	E_CRYO_BIN_CTRL_STATE.ACTIVE_SWITCHING_OFF:
		M_GetStateLabel	:= 'CLOSING...';
	
	E_CRYO_BIN_CTRL_STATE.ERROR:
		M_GetStateLabel	:= 'ERROR';
END_CASE
END_METHOD

METHOD M_SetStatus
VAR_INPUT
	nState:	E_CRYO_BIN_CTRL_STATE;
END_VAR
// Execute the status of the parent FB.
SUPER^.M_SetStatus(nState);


// Handle alarms
M_UpdateAlarms();
END_METHOD

METHOD M_UpdateAlarms
VAR_INPUT
END_VAR
VAR
	stEventEntry : TcEventEntry;
	sText : STRING;
END_VAR
// Array of EventEntry is initialised in the M_Configure method with 
// the alarms defined for the Valve.

fbAlarmHandler(stAlarms := stat.stAlarms);


// Trigger alarms in case of failure.
// The alarms are raised with a rising edge trigger.
// The alarms are cleared with a falling edge trigger.
IF stat.nState = E_CRYO_BIN_CTRL_STATE.ERROR THEN
	IF Actuator.i_nCouplerState <> 8 THEN
		// System not OPERATIONAL or
		// i_nCouplerState not linked to State variable.
		fbAlarmHandler.M_SetAlarm(Tc_Events.CryoValveEventClass.HardwareError);
		stat.sState	:= 'ERROR: System not OPERATIONAL';
	ELSIF Actuator.stat.nLastCommand = E_CRYO_BIN_ACT_CMD.OFF	THEN
		// Valve failed to Close.
		fbAlarmHandler.M_SetAlarm(Tc_Events.CryoValveEventClass.FailureClose);
		stat.sState	:= 'ERROR: Valve failed to CLOSE.';
	ELSIF Actuator.stat.nLastCommand = E_CRYO_BIN_ACT_CMD.ON	THEN
		// Valve failed to Open.
		fbAlarmHandler.M_SetAlarm(Tc_Events.CryoValveEventClass.FailureOpen);
		stat.sState	:= 'ERROR: Valve failed to OPEN.';
	END_IF

END_IF

//
// Clear non-active alarms
// Alarms and their indexes are defined in M_Configure().
// There are three alarms for Valves:
//   0: NOT_OP
//   1: CLOSE failed
//   2: OPEN  failed
//
IF fbAlarmHandler.arrAlarmState[0]  AND  Actuator.i_nCouplerState = 8 THEN
	fbAlarmHandler.M_ClearAlarm(Tc_Events.CryoValveEventClass.HardwareError);
END_IF

IF fbAlarmHandler.arrAlarmState[1]  AND  stat.nState <> E_CRYO_BIN_CTRL_STATE.ERROR THEN
	fbAlarmHandler.M_ClearAlarm(Tc_Events.CryoValveEventClass.FailureClose);
END_IF

IF fbAlarmHandler.arrAlarmState[2] = TRUE  AND  stat.nState <> E_CRYO_BIN_CTRL_STATE.ERROR THEN
	fbAlarmHandler.M_ClearAlarm(Tc_Events.CryoValveEventClass.FailureOpen);
END_IF


fbAlarmHandler.M_ProcessAlarms(
	arrEventEntry := arrEventEntry,
	sEventString := in_sName);
END_METHOD

METHOD M_User_SetAction : INT
VAR_INPUT
END_VAR
// TODO USER
// Set Valve command based on the input parameter in_bEnable.
//
	
IF	stat.nState = E_CRYO_BIN_CTRL_STATE.ACTIVE_OFF  AND in_bEnable THEN
	// Activate the actuator, i.e. open the valve
	M_User_SetAction	:= E_CRYO_BIN_CTRL_ACTION.ON;
ELSIF  stat.nState = E_CRYO_BIN_CTRL_STATE.ACTIVE_ON AND NOT in_bEnable THEN
	// Dectivate the actuator, i.e. close the valve
	M_User_SetAction	:= E_CRYO_BIN_CTRL_ACTION.OFF;
ELSE
	// Don't do anything
	M_User_SetAction	:= E_CRYO_BIN_CTRL_ACTION.NONE;
END_IF
END_METHOD

END_FUNCTION_BLOCK

// ---- POUs/Valve/FB_CRYO_BIN_CTRL.TcPOU
// Binary Controller
FUNCTION_BLOCK FB_CRYO_BIN_CTRL
VAR_INPUT
	in_sName:			STRING := 'Binary Controller';	// Controller name
	in_nFeedback:		E_CRYO_BIN_ACT_FEEDBACK := E_CRYO_BIN_ACT_FEEDBACK.ON_ONLY;	// Feedbacks
	in_nTimeout:		UDINT := 10000;	// Timeout for switching on/off [ms]. Default 10000.
	in_bActiveLowCtrl:	BOOL := FALSE;	// Active Low for Control output
	in_bActiveLowStat:	BOOL := FALSE;	// Active Low for Status signals, i.e. feedback
	in_bEnable:			BOOL := FALSE;	// Controller active while in_bEnable is TRUE
END_VAR
VAR
	
	{attribute 'OPC.UA.DA' := '1'}
	Actuator:	FB_CRYO_BIN_ACT;	// Heater, valve, etc.
	
	{attribute 'OPC.UA.DA' := '1'}
	{attribute 'OPC.UA.DA.Access' := '1'}
	stat:		T_CRYO_BIN_CTRL_STATUS;


	{attribute 'OPC.UA.DA' := '0'}
	bReset:		BOOL := FALSE;		// RESET Command


	{attribute 'OPC.UA.DA' := '0'}
	timer:		TON;		// Timer for commands
	
	// Controller logs
	logs:	FB_CRYO_FUNCTION_LOG;
	
	//
	// Triggers.
	//
	// Capture Enable/Disable.
	trigEnable:		R_TRIG;	// in_bEnable
	trigDisable:	F_TRIG;	// in_bEnable
	// Capture ON/OFF.
	trigON:			R_TRIG;	// i_bIn
	trigOFF:		F_TRIG;	// i_bIn
END_VAR

// Don't do anything until the controller is configured
IF NOT stat.bConfigured THEN
	M_Configure();
	RETURN;
END_IF

// Increment cycle counter
stat.nCycleCounter := stat.nCycleCounter + 1;


// Execute Actuator FB on every cycle
Actuator(
	in_nFeedback		:= in_nFeedback,
	in_nTimeout			:= in_nTimeout,
	in_bActiveLowCtrl	:= in_bActiveLowCtrl,
	in_bActiveLowStat	:= in_bActiveLowStat);


CASE stat.nState OF
	/////////////////////////////////
	E_CRYO_BIN_CTRL_STATE.NONE:
	/////////////////////////////////
	//
	// This is the state on power-up.
	// Determine the initial state based on the command amd actuator state.
	IF Actuator.stat.bError  OR NOT stat.bCtrlOK	THEN
		stat.nState	:= E_CRYO_BIN_CTRL_STATE.ERROR;
	ELSIF in_bEnable  AND  Actuator.stat.bON	THEN
		stat.nState	:= E_CRYO_BIN_CTRL_STATE.ACTIVE_ON;
	ELSIF in_bEnable  AND  Actuator.stat.bOFF	THEN
		stat.nState	:= E_CRYO_BIN_CTRL_STATE.ACTIVE_OFF;
	ELSIF NOT in_bEnable  THEN
		stat.nState	:= E_CRYO_BIN_CTRL_STATE.OFF;
	END_IF
	M_SetStatus(stat.nState);	
	logs.M_LogInfo(M_GetStateLabel(stat.nState));
	RETURN;
	

	/////////////////////////////////
	E_CRYO_BIN_CTRL_STATE.OFF:
	/////////////////////////////////
	//
	IF	Actuator.stat.bError	OR NOT stat.bCtrlOK	THEN
		stat.nState	:= E_CRYO_BIN_CTRL_STATE.ERROR;
	ELSIF in_bEnable  THEN
		// Activate the control loop.
		// Goto Active_Off first.
		//
		// Start the timer
		timer(IN:=FALSE);
		timer(IN:=TRUE, PT:=UDINT_TO_TIME(in_nTimeout));
		// Set next state
		stat.nState	:= E_CRYO_BIN_CTRL_STATE.ACTIVE_OFF;
	END_IF
	M_SetStatus(stat.nState);	
	RETURN;
	
	
	/////////////////////////////////
	E_CRYO_BIN_CTRL_STATE.ACTIVE_OFF:
	/////////////////////////////////
	//
	IF	Actuator.stat.bError	OR NOT stat.bCtrlOK  THEN
		stat.nState	:= E_CRYO_BIN_CTRL_STATE.ERROR;
	ELSIF NOT in_bEnable  THEN
		// Goto Off.
		//
		// Set next state
		stat.nState	:= E_CRYO_BIN_CTRL_STATE.OFF;
	ELSIF M_User_SetAction() = E_CRYO_BIN_CTRL_ACTION.ON THEN
		// Goto Active_Off.
		//
		// Start the timer
		timer(IN:=FALSE);
		timer(IN:=TRUE, PT:=UDINT_TO_TIME(in_nTimeout));
		
		// Trigger action
		Actuator(in_bExecute:=FALSE);
		Actuator(in_bExecute:=TRUE, in_nCommand:=E_CRYO_BIN_ACT_CMD.ON);
		
		// Set next state
		stat.nState	:= E_CRYO_BIN_CTRL_STATE.ACTIVE_SWITCHING_ON;
		logs.M_LogInfo(M_GetStateLabel(stat.nState));
	END_IF
	M_SetStatus(stat.nState);	
	RETURN;
	
	
	//////////////////////////////////////////
	E_CRYO_BIN_CTRL_STATE.ACTIVE_SWITCHING_ON:
	//////////////////////////////////////////
	//
	// Check for timeout
	timer(IN:=TRUE);
	IF timer.Q THEN
		// Stop the timer
		timer(IN:=FALSE);
		// Goto ERROR state
		stat.nState	:= E_CRYO_BIN_CTRL_STATE.ERROR;
	ELSIF	Actuator.stat.bError	THEN
		stat.nState	:= E_CRYO_BIN_CTRL_STATE.ERROR;
	ELSIF Actuator.stat.bON THEN
		// The actuator is ON, transition completed.
		// Goto Active_On.
		stat.nState	:= E_CRYO_BIN_CTRL_STATE.ACTIVE_ON;
		logs.M_LogInfo(M_GetStateLabel(stat.nState));
	END_IF
	M_SetStatus(stat.nState);	
	RETURN;
	

	/////////////////////////////////
	E_CRYO_BIN_CTRL_STATE.ACTIVE_ON:
	/////////////////////////////////
	//
	IF	Actuator.stat.bError	THEN
		stat.nState	:= E_CRYO_BIN_CTRL_STATE.ERROR;
	ELSIF	NOT in_bEnable 		OR  
			NOT stat.bCtrlOK	OR
			M_User_SetAction() = E_CRYO_BIN_CTRL_ACTION.OFF THEN
		// Goto Active_Off.
		// If NOT in_bExecute, the system will continue to complete OFF
		//
		// Start the timer
		timer(IN:=FALSE);
		timer(IN:=TRUE, PT:=UDINT_TO_TIME(in_nTimeout));
		
		// Trigger action
		Actuator(in_bExecute:=FALSE);
		Actuator(in_bExecute:=TRUE, in_nCommand:=E_CRYO_BIN_ACT_CMD.OFF);
		
		// Set next state
		stat.nState	:= E_CRYO_BIN_CTRL_STATE.ACTIVE_SWITCHING_OFF;
		logs.M_LogInfo(M_GetStateLabel(stat.nState));
	END_IF
	M_SetStatus(stat.nState);	
	RETURN;
	
	
	///////////////////////////////////////////
	E_CRYO_BIN_CTRL_STATE.ACTIVE_SWITCHING_OFF:
	///////////////////////////////////////////
	//
	// Check for timeout
	timer(IN:=TRUE);
	IF timer.Q THEN
		// Stop the timer
		timer(IN:=FALSE);
		// Goto ERROR state
		stat.nState	:= E_CRYO_BIN_CTRL_STATE.ERROR;
	ELSIF	Actuator.stat.bError	THEN
		stat.nState	:= E_CRYO_BIN_CTRL_STATE.ERROR;
	ELSIF Actuator.stat.bOFF THEN
		// The actuator is OFF, transition completed.
		// Goto Active_Off.
		stat.nState	:= E_CRYO_BIN_CTRL_STATE.ACTIVE_OFF;
		logs.M_LogInfo(M_GetStateLabel(stat.nState));
	END_IF
	M_SetStatus(stat.nState);	
	RETURN;
	
	/////////////////////////////////
	E_CRYO_BIN_CTRL_STATE.ERROR:
	/////////////////////////////////
	//
	M_User_TryRecovery();

END_CASE

METHOD M_Configure
VAR_INPUT
END_VAR
// Overwrite this method for specific implementation.
// Here we have just a dummy implementation to set
// stat.bConfigured	:= TRUE;


// Device specific implementation
// TODO


// A MUST !!!

// This call just configures logs at the very start.
// Logging is done by explicit calls to M_LogInfo().
logs(in_sName := in_sName);

stat.bConfigured	:= TRUE;
END_METHOD

// Set labels for logging.
// Examples:
//	ON, OFF (for heaters)
//	OPEN, CLOSE (for valves)
METHOD M_GetStateLabel : STRING
VAR_INPUT
	state:	E_CRYO_BIN_CTRL_STATE;
END_VAR
CASE state OF
	E_CRYO_BIN_CTRL_STATE.OFF:
		M_GetStateLabel	:= 'OFF';
	
	E_CRYO_BIN_CTRL_STATE.ACTIVE_SWITCHING_ON:
		M_GetStateLabel	:= 'SWITCHING_ON';
	
	E_CRYO_BIN_CTRL_STATE.ACTIVE_OFF:
		M_GetStateLabel	:= 'OFF';
	
	E_CRYO_BIN_CTRL_STATE.ACTIVE_ON:
		M_GetStateLabel	:= 'ON';
	
	E_CRYO_BIN_CTRL_STATE.ACTIVE_SWITCHING_OFF:
		M_GetStateLabel	:= 'SWITCHING_OFF';
	
	E_CRYO_BIN_CTRL_STATE.ERROR:
		M_GetStateLabel	:= 'ERROR';
END_CASE
END_METHOD

METHOD M_Reset
VAR_INPUT
END_VAR
// By setting the bReset flag,
// The actuator will try to exit error state.
// In ERROR state, method M_User_TryRecovery() is executed.
bReset	:= TRUE;
END_METHOD

METHOD M_SetStatus
VAR_INPUT
	nState:	E_CRYO_BIN_CTRL_STATE;
END_VAR
stat.bActON		:= Actuator.stat.bON;
stat.bActOFF	:= Actuator.stat.bOFF;


CASE nState OF
	
	E_CRYO_BIN_CTRL_STATE.OFF:
	stat.bDone	:= TRUE;
	stat.bBusy	:= FALSE;
	stat.bError	:= FALSE;
	stat.bActive:= FALSE;
	stat.sState	:= 'OFF';
	
	E_CRYO_BIN_CTRL_STATE.ACTIVE_OFF:
	stat.bDone	:= TRUE;
	stat.bBusy	:= FALSE;
	stat.bError	:= FALSE;
	stat.bActive:= TRUE;
	stat.sState	:= 'ACTIVE_OFF';
	
	E_CRYO_BIN_CTRL_STATE.ACTIVE_ON:
	stat.bDone	:= TRUE;
	stat.bBusy	:= FALSE;
	stat.bError	:= FALSE;
	stat.bActive:= TRUE;
	stat.sState	:= 'ACTIVE_ON';
	
	E_CRYO_BIN_CTRL_STATE.ACTIVE_SWITCHING_ON:
	stat.bDone	:= FALSE;
	stat.bBusy	:= TRUE;
	stat.bError	:= FALSE;
	stat.bActive:= TRUE;
	stat.sState	:= 'ACTIVE_SWITCHING_ON...';
	
	E_CRYO_BIN_CTRL_STATE.ACTIVE_SWITCHING_OFF:
	stat.bDone	:= FALSE;
	stat.bBusy	:= TRUE;
	stat.bError	:= FALSE;
	stat.bActive:= TRUE;
	stat.sState	:= 'ACTIVE_SWITCHING_OFF...';
	
	E_CRYO_BIN_CTRL_STATE.ERROR:
	stat.bDone	:= TRUE;
	stat.bBusy	:= FALSE;
	stat.bError	:= TRUE;
	stat.bActive:= FALSE;
	stat.sState	:= 'ERROR';

END_CASE
END_METHOD

METHOD M_User_SetAction : INT
VAR_INPUT
END_VAR
// TODO USER
//
// This method implements the logic for controlling the actuator.
// The actuator can be a heater, valve, etc.
//
// This example implements the heater control with the following assumptions:
// There are two input values from sensors and two deltas for comparison.
//
// in_lrInput1 - Temperature of the Cryo Bench (B)
// in_lrInput2 - Temperature of the Detector (D). Coming from Lakeshore.
// in_lrPar1 - Delta [K] to turn the heater ON:  IF B < D - in_lrPar1
// in_lrPar2 - Delta [K] to turn the heater OFF: IF B > D - in_lrPar2
//
// in_lrDelta1 > in_lrDelta2, e.g. 10K > 4K.
//
IF	stat.nState = E_CRYO_BIN_CTRL_STATE.ACTIVE_OFF  OR  
	stat.nState = E_CRYO_BIN_CTRL_STATE.ACTIVE_ON THEN
(*	
	IF in_lrInput1 < in_lrInput2 - in_lrPar1 THEN
		// Activate the actuator
		M_User_SetOutput	:= E_CRYO_BIN_CTRL_ACTION.ON;
	ELSIF in_lrInput1 > in_lrInput2 - in_lrPar2 THEN
		// Dectivate the actuator
		M_User_SetOutput	:= E_CRYO_BIN_CTRL_ACTION.OFF;
	END_IF
*)
ELSE
	// Don't do anything
	M_User_SetAction	:= E_CRYO_BIN_CTRL_ACTION.NONE;
END_IF
END_METHOD

METHOD M_User_TryRecovery
VAR_INPUT
END_VAR
// TODO USER
// This is the default recovery routine.
// To be customided by the user, if needed.
//
IF bReset THEN
	// RESET the controller in order to try to clear error
	bReset	:= FALSE;	// Clear RESET flag
	
	// Start the timer
	timer(IN:=FALSE);
	timer(IN:=TRUE, PT:=T#5S);
	
	// Trigger action
	Actuator(in_bExecute:=FALSE);
	Actuator(in_bExecute:=TRUE, in_nCommand:=E_CRYO_BIN_ACT_CMD.OFF);
	
	// Goto SWITCHING_OFF state
	stat.nState	:= E_CRYO_BIN_CTRL_STATE.ACTIVE_SWITCHING_OFF;
	M_SetStatus(stat.nState);	
ELSIF NOT Actuator.stat.bError AND stat.bCtrlOK  THEN
	// Self recovery since everything seems to be OK now.
	// Goto NONE state.
	// From there proper state will be found and set.
	stat.nState	:= E_CRYO_BIN_CTRL_STATE.NONE;
	M_SetStatus(stat.nState);	
END_IF
END_METHOD

END_FUNCTION_BLOCK

// ---- POUs/Services/FB_SERVICES.TcPOU
FUNCTION_BLOCK FB_SERVICES
VAR_INPUT
END_VAR
VAR_OUTPUT
END_VAR
VAR    
    // Let's always link the EtherCAT DevState, so that 
    // we always have one sync variable (even if all subsystems are disabled)
    {attribute 'TcLinkTo' := 'TIID^Device 1 (EtherCAT)^Inputs^DevState'}
	i_nDevState AT %I* : UINT;
    
    {attribute 'TcLinkTo' := '.i_inTime             := TIID^Device 1 (EtherCAT)^PLC (EK1200)^PTP (EL6688)^  External Sync^Internal time stamp;
                              .i_exTime             := TIID^Device 1 (EtherCAT)^PLC (EK1200)^PTP (EL6688)^  External Sync^External time stamp;
                              .i_dc2TcOffset        := TIID^Device 1 (EtherCAT)^InfoData^DcToTcTimeOffset;
                              .i_dc2ExtOffset       := TIID^Device 1 (EtherCAT)^InfoData^DcToExtTimeOffset;
                              .i_extDevNotConnected := TIID^Device 1 (EtherCAT)^PLC (EK1200)^PTP (EL6688)^  External Sync^External device not connected;
                              .i_AdsAddr            := TIID^Device 1 (EtherCAT)^PLC (EK1200)^PTP (EL6688)^InfoData^AdsAddr;
                              .i_exNtpExtTime       := TIRC^TcCOM Objects^NtpProvider^Outputs^nExtTime;
                              .i_exNtpSysTime       := TIRC^TcCOM Objects^NtpProvider^Outputs^nSysTime;
                              .i_exNtpExtOffset     := TIRC^TcCOM Objects^NtpProvider^Outputs^nSysToExtTimeOffset;
                              .i_NtpConnected       := TIRC^TcCOM Objects^NtpProvider^Diagnostic^bIsConnected;
                              .i_exNtpSynchronized  := TIRC^TcCOM Objects^NtpProvider^Diagnostic^bIsSynchronized'}
    fbTime : FB_TIME;

END_VAR

fbTime();

END_FUNCTION_BLOCK

// ---- HMI/PRG_HMI.TcPOU
{attribute 'OPC.UA.DA' := '0'}
PROGRAM PRG_HMI
VAR
    // System health & busy status
    fbHealthStatus: 		FB_HMI_HEALTH_STATUS;
    fbBusyStatus: 			FB_HMI_BUSY_STATUS;
    fbStatusColor: 			T_HMI_COLORS;
    
    // BUTTONS
    // ===============================================================================================
    
    // buttons at the main screen
    fbHomeButton: 			FB_HMI_BUTTON('Home'     , 		'Start'      , 	E_HMI_TABS.HOME);
    fbServicesButton : 		FB_HMI_BUTTON('Services' , 		'Services'   , 	E_HMI_TABS.SERVICES);	
	fbEventsButton: 		FB_HMI_BUTTON('Events' , 		'Events', 		E_HMI_TABS.EVENTS);
	fbCryoInterlocksButton: FB_HMI_BUTTON('Cryo Interlocks' ,'Interlock', 	E_HMI_TABS.CRYO_INTERLOCKS);
	
	// ICS Subsystem buttons
	fbShuttersButton: 		FB_HMI_BUTTON('Shutters' , 		'', 			E_HMI_TABS.SHUTTERS);
	fbTipTiltButton: 		FB_HMI_BUTTON('Tip Tilt' , 		'', 			E_HMI_TABS.TIP_TILT);
	fbDelayLinesButton: 	FB_HMI_BUTTON('Delay Lines' , 	'', 			E_HMI_TABS.DELAY_LINES);
	fbCO2TransStagesButton: FB_HMI_BUTTON('CO2 Translation','', 			E_HMI_TABS.CO2_TRANSLATION_STAGES);
	fbZnSeActuatorsButton: 	FB_HMI_BUTTON('ZnSe Actuators' ,'', 			E_HMI_TABS.ZNSE_ACTUATORS);
	fbBirefringenceButton: 	FB_HMI_BUTTON('Birefringence' , '', 			E_HMI_TABS.BIREFRINGENCE_ACTUATORS);
	fbBeamSplitterButton: 	FB_HMI_BUTTON('Beam Splitter' , '', 			E_HMI_TABS.CALIBRATION_UNIT_BEAM_SPLITER);
	fbCO2PressureButton: 	FB_HMI_BUTTON('CO2 Pressure' , 	'', 			E_HMI_TABS.CO2_PRESSURE_CONTROL);
	
    // COMPONENTS
    // ===============================================================================================

    {attribute 'OPC.UA.DA' := '0'}
    fbServices: 			FB_HMI_SERVICES;
	{attribute 'OPC.UA.DA' := '0'}
	fbEvents: 				FB_HMI_EVENTS;
	{attribute 'OPC.UA.DA' := '0'}
	fbCryoInterlocks: 		FB_HMI_CRYO_INTERLOCKS;
	
	{attribute 'OPC.UA.DA' := '0'}
	fbShutters:				FB_HMI_SHUTTERS;
	{attribute 'OPC.UA.DA' := '0'}	
	fbTipTilt:				FB_HMI_TIP_TILT;
	{attribute 'OPC.UA.DA' := '0'}
	fbDelayLines:	        FB_HMI_DELAY_LINES;
	{attribute 'OPC.UA.DA' := '0'}
	fbCO2TransStages:       FB_HMI_CO2_TRANS_STAGES;
	{attribute 'OPC.UA.DA' := '0'}
	fbZnSeActuators:        FB_HMI_ZNSE_ACTUATORS;
	{attribute 'OPC.UA.DA' := '0'}
	fbBirefringence:	    FB_HMI_BIREFRINGENCE;
	{attribute 'OPC.UA.DA' := '0'}
	fbBeamSplitter:         FB_HMI_CALIBRATION_BEAM_SPLITTER;
	{attribute 'OPC.UA.DA' := '0'}
	fbCO2Pressure:          FB_HMI_CO2_PRESSURE_CONTROL;

    
    // active tab of the main frame
    eActiveTab : E_HMI_TABS := E_HMI_TABS.HOME;
    sActiveName : STRING;
END_VAR

//// update the components
fbServices(fbInstance := MAIN.fbServices);
fbEvents(); 				
fbCryoInterlocks(fbInstance := MAIN.nott_ics.Cryo_Interlocks); 		

// SubSystems
fbShutters(fbInstance := MAIN.nott_ics.Shutters);			
fbTipTilt(fbInstance := MAIN.nott_ics.TipTilt);		
fbDelayLines(fbInstance := MAIN.nott_ics.Delay_Lines);			
fbCO2TransStages(fbInstance := MAIN.nott_ics.CO2TransStages);					
fbZnSeActuators(fbInstance := MAIN.nott_ics.ZnSeActuators);	 		
fbBirefringence(fbInstance := MAIN.nott_ics.Birefringence);		
fbBeamSplitter(fbInstance := MAIN.nott_ics.Calibration_Unit_Beam_Splitter);				
fbCO2Pressure(fbInstance := MAIN.nott_ics.CO2_Pressure_Control);

// update the status
M_UpdateStatus();

// update the system-level buttons
fbHomeButton(stColor := fbStatusColor, nActiveTab := eActiveTab, sActiveName := sActiveName);
// buttons at the main screen 
fbServicesButton(stColor := fbServices.fbStatusColor, nActiveTab := eActiveTab, sActiveName := sActiveName);	
fbEventsButton(stColor:= fbEvents.fbStatusColor, nActiveTab:= eActiveTab, sActiveName:= sActiveName);		
fbCryoInterlocksButton(stColor:= fbCryoInterlocks.fbStatusColor, nActiveTab:= eActiveTab, sActiveName:= sActiveName); 	

fbShuttersButton(stColor:= fbShutters.fbStatusColor, nActiveTab:= eActiveTab, sActiveName:= sActiveName); 			
fbTipTiltButton(stColor:= fbTipTilt.fbStatusColor, nActiveTab:= eActiveTab, sActiveName:= sActiveName); 		
fbDelayLinesButton(stColor:= fbDelayLines.fbStatusColor, nActiveTab:= eActiveTab, sActiveName:= sActiveName); 	
fbCO2TransStagesButton(stColor:= fbCO2TransStages.fbStatusColor, nActiveTab:= eActiveTab, sActiveName:= sActiveName); 				
fbZnSeActuatorsButton(stColor:= fbZnSeActuators.fbStatusColor, nActiveTab:= eActiveTab, sActiveName:= sActiveName); 		
fbBirefringenceButton(stColor:= fbBirefringence.fbStatusColor, nActiveTab:= eActiveTab, sActiveName:= sActiveName); 		
fbBeamSplitterButton(stColor:= fbBeamSplitter.fbStatusColor, nActiveTab:= eActiveTab, sActiveName:= sActiveName); 			
fbCO2PressureButton(stColor:= fbCO2Pressure.fbStatusColor, nActiveTab:= eActiveTab, sActiveName:= sActiveName);

METHOD M_UpdateStatus
VAR_INPUT
END_VAR
// update the health & busy statuses
//fbHealthStatus(
//    bIsEnabled :=   fbImg.fbHealthStatus.bEnabled
//                AND fbSca.fbHealthStatus.bEnabled,
//    bIsGood :=      fbImg.fbHealthStatus.bGood
//                AND fbSca.fbHealthStatus.bGood);
              //AND fbServices.fbHealthStatus.bGood
              //AND fbLms.fbHealthStatus.bGood (* AND ... *));
//fbBusyStatus(
//    bIsEnabled :=   fbImg.fbBusyStatus.bEnabled
//                AND fbSca.fbBusyStatus.bEnabled,
//    bIsBusy := fbServices.fbBusyStatus.bBusy 
//                 OR fbImg.fbBusyStatus.bBusy 
//                 OR fbLms.fbBusyStatus.bBusy 
//                 OR fbSca.fbBusyStatus.bBusy);

fbStatusColor := F_HMI_HEALTH_BUSY_TO_COLOR(fbHealthStatus, fbBusyStatus);
END_METHOD

END_PROGRAM

// ---- HMI/POUs/Services/Status/FB_HMI_HEALTH_STATUS.TcPOU
FUNCTION_BLOCK FB_HMI_HEALTH_STATUS
VAR_INPUT
	// TRUE if the subject is in Good health
	bIsGood: BOOL;
	// TRUE to add a warning to the Good health state
	bHasWarning: BOOL := FALSE;
	// TRUE if the health status is used
	bIsEnabled: BOOL := TRUE;
END_VAR
VAR_OUTPUT
	// TRUE if the subject is enabled
	bEnabled: BOOL;
    // TRUE if the subject is in good health
	bGood: BOOL;
	// TRUE if the subject is in good health, but there are one or more warnings present
	bWarning: BOOL;
	// TRUE if the subject is in bad health
	bBad: BOOL;
END_VAR
VAR_IN_OUT
END_VAR
VAR
END_VAR

bEnabled := bIsEnabled;
bBad := (NOT(bIsGood)) AND bIsEnabled;
bGood := (bIsGood AND (NOT(bHasWarning))) AND bIsEnabled;
bWarning := (bIsGood AND bHasWarning) AND bIsEnabled;

END_FUNCTION_BLOCK

// ---- HMI/POUs/Services/Status/FB_HMI_BUSY_STATUS.TcPOU
FUNCTION_BLOCK FB_HMI_BUSY_STATUS
VAR_INPUT
	// TRUE if busy
	bIsBusy: BOOL;
	// TRUE if the busy status is used
	bIsEnabled: BOOL := TRUE;
END_VAR
VAR_OUTPUT
	// TRUE if the subject is enabled
	bEnabled: BOOL;
	///The subject is idle
	bIdle: BOOL;
	///The subject is busy
	bBusy: BOOL;
END_VAR
VAR_IN_OUT
END_VAR
VAR
END_VAR

bBusy := bIsBusy AND bIsEnabled;
bIdle := (NOT(bIsBusy)) AND bIsEnabled;

END_FUNCTION_BLOCK

// ---- HMI/POUs/Util/Button/FB_HMI_BUTTON.TcPOU
FUNCTION_BLOCK FB_HMI_BUTTON
VAR_INPUT
    stColor : T_HMI_COLORS;
END_VAR
VAR_IN_OUT
    nActiveTab : INT;
    sActiveName : STRING;
END_VAR
VAR_OUTPUT
    sName : STRING;
    sIconName : STRING;
    nThisTab : INT;
    bActivated : BOOL;
    bNotActivated : BOOL;
    
    bIsNotGreen : BOOL;
    bIsNotRed : BOOL;
    bIsNotBlue : BOOL;
    bIsNotOrange : BOOL;
    bIsNotGray : BOOL;
END_VAR
VAR
    bDoActivate : BOOL;
    bPreviouslyActive : BOOL;
END_VAR

IF bDoActivate THEN
    nActiveTab := nThisTab;
    bDoActivate := FALSE;
END_IF

bActivated := nActiveTab = nThisTab;
bNotActivated := NOT bActivated;

IF bActivated AND NOT bPreviouslyActive THEN
    sActiveName := sName;
    bPreviouslyActive := TRUE;
END_IF

IF bNotActivated THEN
    bPreviouslyActive := FALSE;
END_IF

bIsNotRed    := stColor.bg <> E_HMI_Colors.RED;
bIsNotBlue   := stColor.bg <> E_HMI_Colors.BLUE;
bIsNotOrange := stColor.bg <> E_HMI_Colors.ORANGE;
bIsNotGray   := stColor.bg <> E_HMI_Colors.GRAY;
bIsNotGreen  := stColor.bg <> E_HMI_Colors.GREEN;

METHOD FB_init : BOOL
VAR_INPUT
	bInitRetains : BOOL; // if TRUE, the retain variables are initialized (warm start / cold start)
	bInCopyCode : BOOL;  // if TRUE, the instance afterwards gets moved into the copy code (online change)
    sName : STRING;
    sIconName : STRING;
    nThisTab : INT;
END_VAR
THIS^.sName := sName;
THIS^.sIconName := sIconName;
THIS^.nThisTab := nThisTab;
END_METHOD

METHOD M_SetIconName
VAR_INPUT
    sIconName : STRING;
END_VAR
THIS^.sIconName := sIconName;
END_METHOD

END_FUNCTION_BLOCK

// ---- HMI/POUs/Services/FB_HMI_SERVICES.TcPOU
FUNCTION_BLOCK FB_HMI_SERVICES EXTENDS FB_HMI_COMPONENT
VAR_INPUT
END_VAR
VAR_OUTPUT
END_VAR
VAR_IN_OUT
    fbInstance : FB_SERVICES;
END_VAR
VAR
    fbTime : FB_HMI_SERVICES_TIME;
END_VAR

fbTime(fbInstance := fbInstance.fbTime);

fbHealthStatus(
    bIsEnabled  := fbTime.fbHealthStatus.bEnabled,
    bIsGood     := fbTime.fbHealthStatus.bGood);
fbBusyStatus(
    bIsEnabled  := fbTime.fbBusyStatus.bEnabled,
    bIsBusy     := fbTime.fbBusyStatus.bBusy);

M_UpdateStatusColor();

END_FUNCTION_BLOCK

// ---- HMI/POUs/Util/Component/FB_HMI_COMPONENT.TcPOU
FUNCTION_BLOCK FB_HMI_COMPONENT
VAR_INPUT
END_VAR
VAR_OUTPUT
    fbHealthStatus : FB_HMI_HEALTH_STATUS;
    fbBusyStatus : FB_HMI_BUSY_STATUS;
    fbStatusColor : T_HMI_COLORS;
END_VAR
VAR
END_VAR

METHOD PROTECTED M_UpdateStatusColor
VAR_INPUT
END_VAR
// health and busy states must be updated by the subtype before calling this method!
fbStatusColor := F_HMI_HEALTH_BUSY_TO_COLOR(fbHealthStatus, fbBusyStatus);
END_METHOD

END_FUNCTION_BLOCK

// ---- HMI/POUs/Services/Status/F_HMI_HEALTH_BUSY_TO_COLOR.TcPOU
FUNCTION F_HMI_HEALTH_BUSY_TO_COLOR : T_HMI_COLORS
VAR_IN_OUT
    fbHealthStatus : FB_HMI_HEALTH_STATUS;
    fbBusyStatus   : FB_HMI_BUSY_STATUS;
END_VAR
VAR_OUTPUT
END_VAR
VAR
END_VAR

IF fbHealthStatus.bGood THEN
	IF fbBusyStatus.bBusy THEN
		F_HMI_HEALTH_BUSY_TO_COLOR.fg := E_HMI_COLORS.WHITE;
		F_HMI_HEALTH_BUSY_TO_COLOR.bg := E_HMI_COLORS.BLUE;
	ELSE
		F_HMI_HEALTH_BUSY_TO_COLOR.fg := E_HMI_COLORS.BLACK;
		F_HMI_HEALTH_BUSY_TO_COLOR.bg := E_HMI_COLORS.GREEN;
	END_IF
ELSIF fbHealthStatus.bBad THEN
	F_HMI_HEALTH_BUSY_TO_COLOR.fg := E_HMI_COLORS.WHITE;
	F_HMI_HEALTH_BUSY_TO_COLOR.bg := E_HMI_COLORS.RED;
ELSIF fbHealthStatus.bWarning THEN
	F_HMI_HEALTH_BUSY_TO_COLOR.fg := E_HMI_COLORS.WHITE;
	F_HMI_HEALTH_BUSY_TO_COLOR.bg := E_HMI_COLORS.ORANGE;
ELSE
	F_HMI_HEALTH_BUSY_TO_COLOR.fg := E_HMI_COLORS.BLACK;
	F_HMI_HEALTH_BUSY_TO_COLOR.bg := E_HMI_COLORS.GRAY;
END_IF

END_FUNCTION

// ---- HMI/POUs/Services/FB_HMI_SERVICES_TIME.TcPOU
FUNCTION_BLOCK FB_HMI_SERVICES_TIME EXTENDS FB_HMI_COMPONENT
VAR_INPUT
END_VAR
VAR_OUTPUT
END_VAR
VAR_IN_OUT
    fbInstance : FB_TIME;
END_VAR
VAR
    // because GUI_TEMPLATE_TIME is a large height,
    // and because scrolling doesn't seem to work (bug in TC HMI?),
    // we display the GUI_TEMPLATE_TIME twice, with an offset in between 
    nAbsoluteMovementY : INT := -495;
    
    sUtc : STRING;
END_VAR


// update the health & busy states
fbHealthStatus(
    bIsGood     := fbInstance.stat.signal.qos = E_TIME_SIGNAL_QOS.VALID,
    bIsEnabled  := fbInstance.stat.signal.status = E_TIME_SIGNAL_STATUS.CONNECTED);
fbBusyStatus(bIsBusy := FALSE); // never busy

sUtc := LEFT(fbInstance.stat.sUtcTime, 19); 

M_UpdateStatusColor();

END_FUNCTION_BLOCK

// ---- HMI/POUs/Events/FB_HMI_EVENTS.TcPOU
FUNCTION_BLOCK FB_HMI_EVENTS EXTENDS FB_HMI_COMPONENT
VAR_INPUT
END_VAR
VAR_OUTPUT
END_VAR

END_FUNCTION_BLOCK

// ---- HMI/POUs/CRYO_Interlocks/FB_HMI_CRYO_INTERLOCKS.TcPOU
FUNCTION_BLOCK FB_HMI_CRYO_INTERLOCKS EXTENDS FB_HMI_COMPONENT
VAR_INPUT
END_VAR
VAR_OUTPUT
END_VAR
VAR
END_VAR
VAR_IN_OUT
	{attribute 'OPC.UA.DA' := '0'}
	fbInstance		: FB_NOTT_CRYO_INTERLOCKS;


END_VAR

fbHealthStatus( 
				bIsEnabled:= TRUE, 
				bIsGood := NOT fbInstance.stat.bError,
				bHasWarning := fbInstance.stat.bWarning
				);
				
fbBusyStatus(
				bIsBusy := fbInstance.stat.bBusy,
				bIsEnabled := TRUE);				
M_UpdateStatusColor();

END_FUNCTION_BLOCK

// ---- HMI/POUs/Subsystems/Shutters/FB_HMI_SHUTTERS.TcPOU
FUNCTION_BLOCK FB_HMI_SHUTTERS EXTENDS FB_HMI_COMPONENT
VAR_INPUT
END_VAR
VAR_OUTPUT
END_VAR
VAR
END_VAR
VAR_IN_OUT
	{attribute 'OPC.UA.DA' := '0'}
	fbInstance		: FB_NOTT_SHUTTERS;


END_VAR


fbHealthStatus( 
				bIsEnabled:= TRUE, 
				bIsGood := NOT fbInstance.stat.bError,
				bHasWarning := fbInstance.stat.bWarning
				);
				
fbBusyStatus(
				bIsBusy := fbInstance.stat.bBusy,
				bIsEnabled := TRUE);				
M_UpdateStatusColor();

END_FUNCTION_BLOCK

// ---- HMI/POUs/Subsystems/TipTilt/FB_HMI_TIP_TILT.TcPOU
FUNCTION_BLOCK FB_HMI_TIP_TILT EXTENDS FB_HMI_COMPONENT
VAR_INPUT
END_VAR
VAR_OUTPUT
END_VAR
VAR_IN_OUT
	{attribute 'OPC.UA.DA' := '0'}
	fbInstance		: FB_NOTT_TIP_TILT;
END_VAR
VAR
    // active tab of the main frame
    eActiveTab : E_HMI_TIP_TILT_TABS := E_HMI_TIP_TILT_TABS.TIP_A;
    sActiveName : STRING;
    
    // components
    fbTIPA: 		FB_HMI_TIP_A;
	fbTIPB:			FB_HMI_TIP_B;
	fbTILTA:		FB_HMI_TILT_A;
    fbTILTB: 		FB_HMI_TILT_B;
	

    
    // buttons
    fbTipAButton		: FB_HMI_BUTTON(sName := 'Tip A'         , sIconName := '', nThisTab := E_HMI_TIP_TILT_TABS.TIP_A);
    fbTipBButton        : FB_HMI_BUTTON(sName := 'Tip B'         , sIconName := '', nThisTab := E_HMI_TIP_TILT_TABS.TIP_B);
    fbTiltAButton       : FB_HMI_BUTTON(sName := 'Tilt A'        , sIconName := '', nThisTab := E_HMI_TIP_TILT_TABS.TILT_A);
    fbTiltBButton  		: FB_HMI_BUTTON(sName := 'Tilt B'        , sIconName := '', nThisTab := E_HMI_TIP_TILT_TABS.TILT_B);
    
    // connection status
    sConnected           : STRING;
    eConnectedColor      : E_HMI_COLORS;
END_VAR



// update the components
fbTIPA(fbInstance := fbInstance);
fbTIPB(fbInstance := fbInstance );
fbTILTA(fbInstance := fbInstance );
fbTILTB(fbInstance := fbInstance);

// update the buttons
// sca
fbTipAButton(
    stColor     := fbTIPA.fbStatusColor,
    nActiveTab  := eActiveTab,
    sActiveName := sActiveName);
fbTipBButton(
    stColor     := fbTIPB.fbStatusColor,
    nActiveTab  := eActiveTab,
    sActiveName := sActiveName);
fbTiltAButton(
    stColor     := fbTILTA.fbStatusColor,
    nActiveTab  := eActiveTab,
    sActiveName := sActiveName);
fbTiltBButton(
    stColor     := fbTILTB.fbStatusColor,
    nActiveTab  := eActiveTab,
    sActiveName := sActiveName);


fbHealthStatus( 
				bIsEnabled:= TRUE, 
				bIsGood := NOT fbInstance.stat.bError,
				bHasWarning := fbInstance.stat.bWarning
				);
				
fbBusyStatus(
				bIsBusy := fbInstance.stat.bBusy,
				bIsEnabled := TRUE);
							
M_UpdateStatusColor();

END_FUNCTION_BLOCK

// ---- HMI/POUs/Subsystems/TipTilt/Components/FB_HMI_TIP_A.TcPOU
FUNCTION_BLOCK FB_HMI_TIP_A EXTENDS FB_HMI_COMPONENT
VAR_OUTPUT
END_VAR
VAR_IN_OUT
    fbInstance : FB_NOTT_TIP_TILT;
END_VAR
VAR
END_VAR

fbHealthStatus(

    bIsGood := NOT fbInstance.stat.bError,
    bHasWarning := (    fbInstance.stat.bWarning));
                     
fbBusyStatus(

    bIsBusy := FALSE);

M_UpdateStatusColor();

END_FUNCTION_BLOCK

// ---- HMI/POUs/Subsystems/TipTilt/Components/FB_HMI_TIP_B.TcPOU
FUNCTION_BLOCK FB_HMI_TIP_B EXTENDS FB_HMI_COMPONENT
VAR_OUTPUT
END_VAR
VAR_IN_OUT
    fbInstance : FB_NOTT_TIP_TILT;
END_VAR
VAR
END_VAR

fbHealthStatus(

    bIsGood := NOT fbInstance.stat.bError,
    bHasWarning := (    fbInstance.stat.bWarning));
                     
fbBusyStatus(

    bIsBusy := FALSE);

M_UpdateStatusColor();

END_FUNCTION_BLOCK

// ---- HMI/POUs/Subsystems/TipTilt/Components/FB_HMI_TILT_A.TcPOU
FUNCTION_BLOCK FB_HMI_TILT_A EXTENDS FB_HMI_COMPONENT
VAR_OUTPUT
END_VAR
VAR_IN_OUT
    fbInstance : FB_NOTT_TIP_TILT;
END_VAR
VAR
END_VAR

fbHealthStatus(

    bIsGood := NOT fbInstance.stat.bError,
    bHasWarning := (    fbInstance.stat.bWarning));
                     
fbBusyStatus(
    bIsBusy := FALSE);

M_UpdateStatusColor();

END_FUNCTION_BLOCK

// ---- HMI/POUs/Subsystems/TipTilt/Components/FB_HMI_TILT_B.TcPOU
FUNCTION_BLOCK FB_HMI_TILT_B EXTENDS FB_HMI_COMPONENT
VAR_OUTPUT
END_VAR
VAR_IN_OUT
    fbInstance : FB_NOTT_TIP_TILT;
END_VAR
VAR
END_VAR

fbHealthStatus(

    bIsGood := NOT fbInstance.stat.bError,
    bHasWarning := (    fbInstance.stat.bWarning));
                     
fbBusyStatus(

    bIsBusy := FALSE);

M_UpdateStatusColor();

END_FUNCTION_BLOCK

// ---- HMI/POUs/Subsystems/DelayLines/FB_HMI_DELAY_LINES.TcPOU
FUNCTION_BLOCK FB_HMI_DELAY_LINES EXTENDS FB_HMI_COMPONENT
VAR_INPUT
END_VAR
VAR_OUTPUT
END_VAR
VAR
END_VAR
VAR_IN_OUT
	{attribute 'OPC.UA.DA' := '0'}
	fbInstance		: FB_NOTT_DELAY_LINES;


END_VAR


fbHealthStatus( 
				bIsEnabled:= TRUE, 
				bIsGood := NOT fbInstance.stat.bError,
				bHasWarning := fbInstance.stat.bWarning
				);
				
fbBusyStatus(
				bIsBusy := fbInstance.stat.bBusy,
				bIsEnabled := TRUE);
				
M_UpdateStatusColor();

END_FUNCTION_BLOCK

// ---- HMI/POUs/Subsystems/CO2_Translation_Stages/FB_HMI_CO2_TRANS_STAGES.TcPOU
FUNCTION_BLOCK FB_HMI_CO2_TRANS_STAGES EXTENDS FB_HMI_COMPONENT
VAR_INPUT
END_VAR
VAR_OUTPUT
END_VAR
VAR
END_VAR
VAR_IN_OUT
	{attribute 'OPC.UA.DA' := '0'}
	fbInstance		: FB_NOTT_CO2_TRANS_STAGES;


END_VAR


fbHealthStatus( 
				bIsEnabled:= TRUE, 
				bIsGood := NOT fbInstance.stat.bError,
				bHasWarning := fbInstance.stat.bWarning 
				);
				
fbBusyStatus(
				bIsBusy := fbInstance.stat.bBusy,
				bIsEnabled := TRUE);
				
M_UpdateStatusColor();

END_FUNCTION_BLOCK

// ---- HMI/POUs/Subsystems/ZnSe_Actuators/FB_HMI_ZNSE_ACTUATORS.TcPOU
FUNCTION_BLOCK FB_HMI_ZNSE_ACTUATORS EXTENDS FB_HMI_COMPONENT
VAR_INPUT
END_VAR
VAR_OUTPUT
END_VAR
VAR
END_VAR
VAR_IN_OUT
	{attribute 'OPC.UA.DA' := '0'}
	fbInstance		: FB_NOTT_ZNSE_ACTUATORS;


END_VAR


fbHealthStatus( 
				bIsEnabled:= TRUE, 
				bIsGood := NOT fbInstance.stat.bError,
				bHasWarning := fbInstance.stat.bWarning
				);
				
fbBusyStatus(
				bIsBusy := fbInstance.stat.bBusy,
				bIsEnabled := TRUE);
				
M_UpdateStatusColor();

END_FUNCTION_BLOCK

// ---- HMI/POUs/Subsystems/Birefringence/FB_HMI_BIREFRINGENCE.TcPOU
FUNCTION_BLOCK FB_HMI_BIREFRINGENCE EXTENDS FB_HMI_COMPONENT
VAR_INPUT
END_VAR
VAR_OUTPUT
END_VAR
VAR
END_VAR
VAR_IN_OUT
	{attribute 'OPC.UA.DA' := '0'}
	fbInstance		: FB_NOTT_BIREFRINGENCE;


END_VAR


fbHealthStatus( 
				bIsEnabled:= TRUE, 
				bIsGood := NOT fbInstance.stat.bError,
				bHasWarning := fbInstance.stat.bWarning
				);
				
fbBusyStatus(
				bIsBusy := fbInstance.stat.bBusy,
				bIsEnabled := TRUE);
				
M_UpdateStatusColor();

END_FUNCTION_BLOCK

// ---- HMI/POUs/Subsystems/Beam_Splitter/FB_HMI_CALIBRATION_BEAM_SPLITTER.TcPOU
FUNCTION_BLOCK FB_HMI_CALIBRATION_BEAM_SPLITTER EXTENDS FB_HMI_COMPONENT
VAR_INPUT
END_VAR
VAR_OUTPUT
END_VAR
VAR
END_VAR
VAR_IN_OUT
	{attribute 'OPC.UA.DA' := '0'}
	fbInstance		: FB_NOTT_CALIBRATION_BEAM_SPLITTER;


END_VAR


fbHealthStatus( 
				bIsEnabled:= TRUE, 
				bIsGood := NOT fbInstance.stat.bError,
				bHasWarning := fbInstance.stat.bWarning
				);
				
fbBusyStatus(
				bIsBusy := fbInstance.stat.bBusy,
				bIsEnabled := TRUE);
				
M_UpdateStatusColor();

END_FUNCTION_BLOCK

// ---- HMI/POUs/Subsystems/CO2_Pressure/FB_HMI_CO2_PRESSURE_CONTROL.TcPOU
FUNCTION_BLOCK FB_HMI_CO2_PRESSURE_CONTROL EXTENDS FB_HMI_COMPONENT
VAR_INPUT
END_VAR
VAR_OUTPUT
END_VAR
VAR
END_VAR
VAR_IN_OUT
	{attribute 'OPC.UA.DA' := '0'}
	fbInstance		: FB_NOTT_CO2_PRESSURE_CONTROL;


END_VAR


fbHealthStatus( 
				bIsEnabled:= TRUE, 
				bIsGood := NOT fbInstance.stat.bError,
				bHasWarning := fbInstance.stat.bWarning
				);
				
fbBusyStatus(
				bIsBusy := fbInstance.stat.bBusy,
				bIsEnabled := TRUE);
				
M_UpdateStatusColor();

END_FUNCTION_BLOCK

// ---- HMI/POUs/Devices/Cabinets/FB_HMI_CABINETS.TcPOU
FUNCTION_BLOCK FB_HMI_CABINETS EXTENDS FB_HMI_COMPONENT
VAR_INPUT
END_VAR
VAR_OUTPUT
END_VAR
VAR
END_VAR

END_FUNCTION_BLOCK

// ---- HMI/POUs/Devices/Control_Loops/FB_HMI_CONTROL_LOOPS.TcPOU
FUNCTION_BLOCK FB_HMI_CONTROL_LOOPS EXTENDS FB_HMI_COMPONENT
VAR_INPUT
END_VAR
VAR_OUTPUT
END_VAR
VAR
END_VAR

END_FUNCTION_BLOCK

// ---- HMI/POUs/Devices/Control_Loops/FB_HMI_METIS_CTRL_TEMPERATURE.TcPOU
FUNCTION_BLOCK FB_HMI_METIS_CTRL_TEMPERATURE EXTENDS FB_HMI_COMPONENT
VAR_INPUT
END_VAR
VAR_OUTPUT
END_VAR
VAR_IN_OUT
    fbInstance : FB_METIS_CTRL_TEMPERATURE;
END_VAR
VAR
END_VAR

fbHealthStatus(
    bIsEnabled := fbInstance.cfg.bEnabled,
    bIsGood := fbInstance.stat.bValid);
                     
fbBusyStatus(
    bIsEnabled := FALSE,
    bIsBusy := FALSE);

M_UpdateStatusColor();

END_FUNCTION_BLOCK

// ---- HMI/POUs/Devices/Control_Units/FB_HMI_CONTROL_UNITS.TcPOU
FUNCTION_BLOCK FB_HMI_CONTROL_UNITS EXTENDS FB_HMI_COMPONENT
VAR_INPUT
END_VAR
VAR_OUTPUT
END_VAR
VAR
END_VAR

END_FUNCTION_BLOCK

// ---- HMI/POUs/Devices/Coolers/FB_HMI_COOLERS.TcPOU
FUNCTION_BLOCK FB_HMI_COOLERS EXTENDS FB_HMI_COMPONENT
VAR_INPUT
END_VAR
VAR_OUTPUT
END_VAR
VAR
END_VAR

END_FUNCTION_BLOCK

// ---- HMI/POUs/Devices/Detectors/FB_HMI_DETECTORS.TcPOU
FUNCTION_BLOCK FB_HMI_DETECTORS EXTENDS FB_HMI_COMPONENT
VAR_INPUT
END_VAR
VAR_OUTPUT
END_VAR
VAR
END_VAR

END_FUNCTION_BLOCK

// ---- HMI/POUs/Devices/Heaters/FB_HMI_HEATERS.TcPOU
FUNCTION_BLOCK FB_HMI_HEATERS EXTENDS FB_HMI_COMPONENT
VAR_INPUT
END_VAR
VAR_OUTPUT
END_VAR
VAR
END_VAR

END_FUNCTION_BLOCK

// ---- HMI/POUs/Devices/Heaters/FB_HMI_METIS_HEATER.TcPOU
FUNCTION_BLOCK FB_HMI_METIS_HEATER EXTENDS FB_HMI_COMPONENT
VAR_INPUT
END_VAR
VAR_OUTPUT
END_VAR
VAR_IN_OUT
    fbInstance : FB_METIS_HEATER;
END_VAR
VAR
END_VAR

fbHealthStatus(
    bIsEnabled := fbInstance.stat.bActive,
    bIsGood := NOT fbInstance.stat.bError,
    bHasWarning := fbInstance.stat.bWarning);
                     
fbBusyStatus(
    bIsEnabled := FALSE,
    bIsBusy := FALSE);

M_UpdateStatusColor();

END_FUNCTION_BLOCK

// ---- HMI/POUs/Devices/Lakeshores/FB_HMI_LAKESHORE.TcPOU
FUNCTION_BLOCK FB_HMI_LAKESHORE EXTENDS FB_HMI_COMPONENT
VAR_INPUT
    bConnected : BOOL;
END_VAR
VAR_OUTPUT
END_VAR
VAR_IN_OUT
    fbInstance : FB_METIS_LAKESHORE_336_TCP;
END_VAR
VAR
END_VAR

fbHealthStatus(
    bIsEnabled := bConnected,
    bIsGood := fbInstance.stat.nSubstate = E_RS_BASE_SUBSTATE.OP_MONITORING,
    bHasWarning := fbInstance.stat.bLocal);
                     
fbBusyStatus(
    bIsEnabled := bConnected,
    bIsBusy := fbInstance.stat.nSubstate = E_RS_BASE_SUBSTATE.NOTOP_INITIALIZING);

M_UpdateStatusColor();

END_FUNCTION_BLOCK

// ---- HMI/POUs/Devices/Pressures/FB_HMI_PRESSURES.TcPOU
FUNCTION_BLOCK FB_HMI_PRESSURES EXTENDS FB_HMI_COMPONENT
VAR_INPUT
END_VAR
VAR_OUTPUT
END_VAR
VAR
END_VAR

END_FUNCTION_BLOCK

// ---- HMI/POUs/Devices/Pumps/FB_HMI_PUMPS.TcPOU
FUNCTION_BLOCK FB_HMI_PUMPS EXTENDS FB_HMI_COMPONENT
VAR
	// System health & busy status
//    fbHealthStatus: 		FB_HMI_HEALTH_STATUS;
//    fbBusyStatus: 			FB_HMI_BUSY_STATUS;
//    fbStatusColor: 			T_HMI_COLORS;
	
	// Pumps
	fbRpBranchAButton: 		FB_HMI_BUTTON('RP A' , '', 	E_HMI_PUMPS_TABS.RP_BRANCH_A);
	fbRpBranchBButton: 		FB_HMI_BUTTON('RP B' , '', 	E_HMI_PUMPS_TABS.RP_BRANCH_B);
	fbTpBranchAButton: 		FB_HMI_BUTTON('TP A' , '', 	E_HMI_PUMPS_TABS.TP_BRANCH_A);
	fbTpBranchBButton: 		FB_HMI_BUTTON('TP B' , '', 	E_HMI_PUMPS_TABS.TP_BRANCH_B);
	
		// Pumps
	fbRpBranchA:			FB_HMI_RP_BRANCH_A;
	fbRpBranchB:			FB_HMI_RP_BRANCH_B;
	fbTpBranchA:			FB_HMI_TP_BRANCH_A;
	fbTpBranchB:			FB_HMI_TP_BRANCH_B;
	
	    // active tab of the main frame
    eActiveTab : E_HMI_PUMPS_TABS := E_HMI_PUMPS_TABS.RP_BRANCH_A;
    sActiveName : STRING;

END_VAR


// Pumps
 			
fbRpBranchA();
fbRpBranchB();
fbTpBranchA();
fbTpBranchB();

// Pumps

fbRpBranchAButton(stColor:= fbRpBranchA.fbStatusColor, nActiveTab:= eActiveTab, sActiveName:= sActiveName); 		
fbRpBranchBButton(stColor:= fbRpBranchB.fbStatusColor, nActiveTab:= eActiveTab, sActiveName:= sActiveName); 
fbTpBranchAButton(stColor:= fbTpBranchA.fbStatusColor, nActiveTab:= eActiveTab, sActiveName:= sActiveName); 
fbTpBranchBButton(stColor:= fbTpBranchB.fbStatusColor, nActiveTab:= eActiveTab, sActiveName:= sActiveName);

END_FUNCTION_BLOCK

// ---- HMI/POUs/Devices/Pumps/FB_HMI_RP_BRANCH_A.TcPOU
FUNCTION_BLOCK FB_HMI_RP_BRANCH_A EXTENDS FB_HMI_COMPONENT
VAR_INPUT
END_VAR
VAR_OUTPUT
END_VAR
VAR
END_VAR

END_FUNCTION_BLOCK

// ---- HMI/POUs/Devices/Pumps/FB_HMI_RP_BRANCH_B.TcPOU
FUNCTION_BLOCK FB_HMI_RP_BRANCH_B EXTENDS FB_HMI_COMPONENT
VAR_INPUT
END_VAR
VAR_OUTPUT
END_VAR
VAR
END_VAR

END_FUNCTION_BLOCK

// ---- HMI/POUs/Devices/Pumps/FB_HMI_TP_BRANCH_A.TcPOU
FUNCTION_BLOCK FB_HMI_TP_BRANCH_A EXTENDS FB_HMI_COMPONENT
VAR_INPUT
END_VAR
VAR_OUTPUT
END_VAR
VAR
END_VAR

END_FUNCTION_BLOCK

// ---- HMI/POUs/Devices/Pumps/FB_HMI_TP_BRANCH_B.TcPOU
FUNCTION_BLOCK FB_HMI_TP_BRANCH_B EXTENDS FB_HMI_COMPONENT
VAR_INPUT
END_VAR
VAR_OUTPUT
END_VAR
VAR
END_VAR

END_FUNCTION_BLOCK

// ---- HMI/POUs/Devices/RH/FB_HMI_METIS_RH_SENSOR.TcPOU
FUNCTION_BLOCK FB_HMI_METIS_RH_SENSOR EXTENDS FB_HMI_COMPONENT
VAR_INPUT
END_VAR
VAR_OUTPUT
END_VAR
VAR_IN_OUT
    fbInstance : FB_METIS_RH_SENSOR;
END_VAR
VAR
END_VAR

fbHealthStatus(
    bIsEnabled := fbInstance.stat.bValid,
    bIsGood := NOT fbInstance.stat.bError);

fbBusyStatus(
    bIsEnabled := FALSE,
    bIsBusy := FALSE);

M_UpdateStatusColor();

END_FUNCTION_BLOCK

// ---- HMI/POUs/Devices/Temperatures/Components/FB_HMI_TEMP_VOTERS.TcPOU
FUNCTION_BLOCK FB_HMI_TEMP_VOTERS EXTENDS FB_HMI_COMPONENT
VAR_INPUT
END_VAR
VAR_OUTPUT
END_VAR
VAR_IN_OUT
    fbInstance : FB_METIS_VOTERS;
END_VAR
VAR
    eActiveTab : E_HMI_VOTER_TABS;
    sActiveName : STRING;
    
    fbVoter1Button  : FB_HMI_BUTTON(sName := 'Master' , sIconName := '', nThisTab := E_HMI_VOTER_TABS.VOTER_1);
    fbVoter2Button  : FB_HMI_BUTTON(sName := 'Vot Master 1' , sIconName := '', nThisTab := E_HMI_VOTER_TABS.VOTER_2);
    fbVoter3Button  : FB_HMI_BUTTON(sName := 'Vot Master 2' , sIconName := '', nThisTab := E_HMI_VOTER_TABS.VOTER_3);
    
    
    fbVoter1 : FB_HMI_VOTER;
    fbVoter2 : FB_HMI_VOTER;
    fbVoter3 : FB_HMI_VOTER;
    
END_VAR

fbVoter1(fbInstance := fbInstance.vote_cry_1);
fbVoter2(fbInstance := fbInstance.vote_cry_2);
fbVoter3(fbInstance := fbInstance.vote_cry_3);


fbVoter1Button(stColor := fbVoter1.fbStatusColor, nActiveTab := eActiveTab, sActiveName := sActiveName);
fbVoter2Button(stColor := fbVoter2.fbStatusColor, nActiveTab := eActiveTab, sActiveName := sActiveName);
fbVoter3Button(stColor := fbVoter3.fbStatusColor, nActiveTab := eActiveTab, sActiveName := sActiveName);


fbHealthStatus(
    bIsEnabled :=  fbVoter1.fbHealthStatus.bEnabled
                OR fbVoter2.fbHealthStatus.bEnabled
                OR fbVoter3.fbHealthStatus.bEnabled,
    bIsGood :=  (fbVoter1.fbHealthStatus.bGood OR NOT fbVoter1.fbHealthStatus.bEnabled)
            AND (fbVoter2.fbHealthStatus.bGood OR NOT fbVoter2.fbHealthStatus.bEnabled)
            AND (fbVoter3.fbHealthStatus.bGood OR NOT fbVoter3.fbHealthStatus.bEnabled));

fbBusyStatus(bIsEnabled := FALSE);

M_UpdateStatusColor();

END_FUNCTION_BLOCK

// ---- HMI/POUs/Devices/Voters/FB_HMI_VOTER.TcPOU
FUNCTION_BLOCK FB_HMI_VOTER EXTENDS FB_HMI_COMPONENT
VAR_INPUT
END_VAR
VAR_OUTPUT
END_VAR
VAR_IN_OUT
    fbInstance : FB_METIS_VOTER;
END_VAR
VAR
END_VAR

fbHealthStatus(
    bIsEnabled := fbInstance.stat.bEnabled,
    bIsGood := fbInstance.stat.bValid);
                     
fbBusyStatus(
    bIsEnabled := FALSE,
    bIsBusy := FALSE);

M_UpdateStatusColor();

END_FUNCTION_BLOCK

// ---- HMI/POUs/Devices/Temperatures/FB_HMI_TEMPERATURES.TcPOU
FUNCTION_BLOCK FB_HMI_TEMPERATURES EXTENDS FB_HMI_COMPONENT
VAR_INPUT
END_VAR
VAR_OUTPUT
END_VAR

VAR_IN_OUT
    voters          : FB_METIS_VOTERS;
END_VAR
VAR
    // active tab of the main frame
    eActiveTab : E_HMI_TEMP_TABS := E_HMI_TEMP_TABS.VOTERS;
    sActiveName : STRING;
    
    // components
    fbVoters       		: FB_HMI_TEMP_VOTERS;

    
    // buttons
    fbVotersButton       : FB_HMI_BUTTON(sName := 'Voters'               , sIconName := '', nThisTab := E_HMI_CRY_TABS.VOTERS);

END_VAR

// update the components

fbVoters(fbInstance := voters);

// update the buttons

fbVotersButton(
    stColor     := fbVoters.fbStatusColor,
    nActiveTab  := eActiveTab,
    sActiveName := sActiveName);



// update the summary health/busy status
fbHealthStatus(
    bIsEnabled  := TRUE,
    bIsGood     :=     fbVoters.fbHealthStatus.bGood,
    bHasWarning :=     fbVoters.fbHealthStatus.bWarning);

fbBusyStatus(
    bIsEnabled   := TRUE,
    bIsBusy      :=    fbVoters.fbBusyStatus.bBusy);

M_UpdateStatusColor();

END_FUNCTION_BLOCK

// ---- HMI/POUs/Devices/Valves/FB_HMI_VALVES.TcPOU
FUNCTION_BLOCK FB_HMI_VALVES EXTENDS FB_HMI_COMPONENT
VAR_INPUT
END_VAR
VAR_OUTPUT
END_VAR
VAR
END_VAR

END_FUNCTION_BLOCK

// ---- HMI/POUs/Services/Status/FB_HMI_STATUS.TcPOU
FUNCTION_BLOCK FB_HMI_STATUS
VAR_INPUT
	sText : STRING;
	stColor : T_HMI_COLORS;
END_VAR
VAR_OUTPUT
END_VAR
VAR_IN_OUT
END_VAR
VAR
END_VAR

END_FUNCTION_BLOCK

// ---- HMI/POUs/Services/Status/F_HMI_BUSY_TO_COLOR.TcPOU
FUNCTION F_HMI_BUSY_TO_COLOR : T_HMI_COLORS
VAR_IN_OUT
    fbBusyStatus : FB_HMI_BUSY_STATUS;
END_VAR
VAR_OUTPUT
END_VAR
VAR
END_VAR

IF fbBusyStatus.bIdle THEN
    F_HMI_BUSY_TO_COLOR.fg := E_HMI_COLORS.BLACK;
    F_HMI_BUSY_TO_COLOR.bg := E_HMI_COLORS.GREEN;
ELSIF fbBusyStatus.bBusy THEN
	F_HMI_BUSY_TO_COLOR.fg := E_HMI_COLORS.WHITE;
	F_HMI_BUSY_TO_COLOR.bg := E_HMI_COLORS.BLUE;
ELSE
	F_HMI_BUSY_TO_COLOR.fg := E_HMI_COLORS.BLACK;
	F_HMI_BUSY_TO_COLOR.bg := E_HMI_COLORS.GRAY;
END_IF

END_FUNCTION

// ---- HMI/POUs/Services/Status/F_HMI_HEALTH_TO_COLOR.TcPOU
FUNCTION F_HMI_HEALTH_TO_COLOR : T_HMI_COLORS
VAR_IN_OUT
    fbHealthStatus : FB_HMI_HEALTH_STATUS;
END_VAR
VAR_OUTPUT
END_VAR
VAR
END_VAR

IF fbHealthStatus.bGood THEN
    F_HMI_HEALTH_TO_COLOR.fg := E_HMI_COLORS.BLACK;
    F_HMI_HEALTH_TO_COLOR.bg := E_HMI_COLORS.GREEN;
ELSIF fbHealthStatus.bBad THEN
	F_HMI_HEALTH_TO_COLOR.fg := E_HMI_COLORS.WHITE;
	F_HMI_HEALTH_TO_COLOR.bg := E_HMI_COLORS.RED;
ELSIF fbHealthStatus.bWarning THEN
	F_HMI_HEALTH_TO_COLOR.fg := E_HMI_COLORS.WHITE;
	F_HMI_HEALTH_TO_COLOR.bg := E_HMI_COLORS.ORANGE;
ELSE
	F_HMI_HEALTH_TO_COLOR.fg := E_HMI_COLORS.BLACK;
	F_HMI_HEALTH_TO_COLOR.bg := E_HMI_COLORS.GRAY;
END_IF

END_FUNCTION

// ---- HMI/POUs/Util/Functions/F_GetConnectionColor.TcPOU
FUNCTION F_GetConnectionColor : E_HMI_COLORS
VAR_INPUT
    bConnected : BOOL;
END_VAR
VAR
END_VAR

IF bConnected THEN
    F_GetConnectionColor := E_HMI_COLORS.GREEN;
ELSE
    F_GetConnectionColor := E_HMI_COLORS.RED;
END_IF

END_FUNCTION

// ---- HMI/POUs/Util/Functions/F_GetConnectionString.TcPOU
FUNCTION F_GetConnectionString : STRING
VAR_INPUT
    bConnected : BOOL;
END_VAR
VAR
END_VAR

IF bConnected THEN
    F_GetConnectionString := 'Connected';
ELSE
    F_GetConnectionString := 'Disconnected';
END_IF

END_FUNCTION

// ---- POUs/Functions/F_SysTimeToString.TcPOU
FUNCTION F_SysTimeToString : STRING(23)
VAR_INPUT
	nSysTime : LINT;
END_VAR
VAR
	nFileTime : T_FILETIME;
	
	fbGetSystemTime  : GETSYSTEMTIME;
END_VAR

MEMCPY(ADR(nFileTime), ADR(nSysTime), SIZEOF(nFileTime));


//F_SysTimeToString := DCTIME64_TO_STRING(FILETIME_TO_DCTIME64(nFileTime));


fbGetSystemTime(timeLoDW=>nFileTime.dwLowDateTime, timeHiDW=>nFileTime.dwHighDateTime );
F_SysTimeToString := SYSTEMTIME_TO_STRING( FILETIME_TO_SYSTEMTIME( nFileTime ) );

END_FUNCTION

// ---- POUs/System/FB_NOTT_CRYO_CTRL.TcPOU
FUNCTION_BLOCK FB_NOTT_CRYO_CTRL
VAR_INPUT
END_VAR
VAR_OUTPUT
END_VAR
VAR
	
	temp_1:		FB_CRYO_SENSOR_TEMPERATURE;
	temp_2:		FB_CRYO_SENSOR_TEMPERATURE;
	temp_3:		FB_CRYO_SENSOR_TEMPERATURE;
	temp_4:		FB_CRYO_SENSOR_TEMPERATURE;
	{attribute 'OPC.UA.DA' := '1'}
	lrTempC_1:	LREAL;
	{attribute 'OPC.UA.DA' := '1'}
	lrTempC_2:	LREAL;
	{attribute 'OPC.UA.DA' := '1'}
	lrTempC_3:	LREAL;
	{attribute 'OPC.UA.DA' := '1'}
	lrTempC_4:	LREAL;
END_VAR


M_ReadSensors();

METHOD M_ReadSensors
VAR_INPUT
END_VAR
temp_1(
	in_sName:= 'Temp 1', 
	in_nType:= E_CRYO_SENSOR_TYPE_TEMP.PT100, 
	in_lrScale:= 0.1, 
	in_bIgnoreUnderrange:= TRUE, 
	in_nRampPeriodSec:= 60, 
	in_bResistor_1_64:= );
lrTempC_1 := temp_1.stat.lrTempC;	

temp_2(
	in_sName:= 'Temp 2', 
	in_nType:= E_CRYO_SENSOR_TYPE_TEMP.PT100, 
	in_lrScale:= 0.1, 
	in_bIgnoreUnderrange:= TRUE, 
	in_nRampPeriodSec:= 60, 
	in_bResistor_1_64:= );
lrTempC_2 := temp_2.stat.lrTempC;
	
temp_3(
	in_sName:= 'Temp 3', 
	in_nType:= E_CRYO_SENSOR_TYPE_TEMP.PT100, 
	in_lrScale:= 0.1, 
	in_bIgnoreUnderrange:= TRUE, 
	in_nRampPeriodSec:= 60, 
	in_bResistor_1_64:= );
lrTempC_3 := temp_3.stat.lrTempC;
	
temp_4(
	in_sName:= 'Temp 4', 
	in_nType:= E_CRYO_SENSOR_TYPE_TEMP.PT100, 
	in_lrScale:= 0.1, 
	in_bIgnoreUnderrange:= TRUE, 
	in_nRampPeriodSec:= 60, 
	in_bResistor_1_64:= );
lrTempC_4 := temp_4.stat.lrTempC;
END_METHOD

END_FUNCTION_BLOCK

// ---- GlobalTextList.TcGTLO
TEXTLIST GlobalTextList
  46 = ''
  1904 = '   Ctrl out'
  150 = ' 0 - END [0] [0] (e.g. "END,0,0")'
  151 = ' 1 - Find Index Switch [fast Vel] [slow Vel] (e.g. "FIND_INDEX,10.0,0.5")'
  152 = ' 2 - Find REF Switch Lower Edge [fast Vel] [slow Vel] (e.g. "FIND_REF_LE,8,0.1")'
  135 = ' 3 - Find REF Switch Upper Edge [fast Vel] [slow Vel] (e.g. "FIND_REF_UE,8.5,1")'
  154 = ' 4 - Find Lower HW Limit [fast Vel] [slow Vel] (e.g. "FIND_LHW,5.0,0.2")'
  155 = ' 5 - Find Upper HW Limit [fast Vel] [slow Vel] (e.g. "FIND_UHW,5.0,0.2")'
  160 = ' 6 - Delay [ms] [0] (e.g. "DELAY,3000,0")'
  156 = ' 7 - Move Absolute [vel] [pos] (e.g. "MOVE_ABS,25.0,360.0")'
  157 = ' 8 - Move Relative [vel] [pos] (e.g. "MOVE_REL,25.0,60.0")'
  158 = ' 9 - Calibrate Absolute [pos] [0] (e.g. "CALIB_ABS,180.0,0")'
  671 = '%'
  1501 = '%.0f'
  17 = '%.0f  '
  3988 = '%.1e mbar'
  399 = '%.1f'
  556 = '%.1f '
  3975 = '%.1f %%'
  3934 = '%.1f Hours'
  1371 = '%.1f K'
  5732 = '%.1f min'
  1569 = '%.1f Ohm'
  1115 = '%.1f W'
  1786 = '%.1f °C'
  411 = '%.2f'
  32 = '%.2f  '
  1596 = '%.2f %%'
  930 = '%.2f A'
  196 = '%.2f C'
  273 = '%.2f K'
  559 = '%.2f K/h'
  486 = '%.2f K/min'
  848 = '%.2f °C'
  254 = '%.3e'
  1040 = '%.3e mbar'
  508 = '%.3f'
  1392 = '%.3f s'
  1544 = '%.4e mbar'
  229 = '%.4f'
  3527 = '%.4f K/m'
  992 = '%.5f'
  28 = '%.6f'
  860 = '%.7f'
  1419 = '%.f'
  417 = '%d'
  1270 = '%d ms'
  828 = '%s'
  607 = '%T'
  3257 = '%u'
  1022 = "'Motor.library version'"
  3155 = '(Hours) Refilling cycle time during the Early refilling'
  581 = '(Hours) The total duration of Early Refilling'
  1123 = '(Minutes) LN2 level hold time to reduce oscilations at level change'
  1199 = '+'
  346 = '1'
  5812 = '1. Cryostat Pressure < 1e-4 mbar'
  2053 = '1. Regeneration Safe Temperature Achieved'
  5368 = '1. Vacuum Pumps are OFF'
  4530 = '1. Venting Valves are Closed.'
  710 = '10'
  159 = '10 - Calibrate Relative [pos] [0] (e.g. "CALIB_REL,5.25,0")'
  161 = '11 - Calibrate on Switch [pos] [0.0] (e.g. "CALIB_SWITCH,180.0,0")'
  347 = '2'
  1690 = '2. Evacuation Active'
  3326 = '2. Evacuation Inactive'
  4800 = '2. Warm Up Inactive'
  348 = '3'
  4877 = '3. Cool Down Inactive'
  3916 = '3. Venting Valves Are Closed'
  349 = '4'
  5728 = '4. Regeneration Inactive'
  350 = '5'
  4298 = '5. GN2 Supply Connected'
  3338 = '5. Pumps Are Running'
  186 = '6'
  2726 = '6. All Temperatures > 280 K'
  2949 = '6. LN2 Supply Connected'
  352 = '7'
  353 = '8'
  703 = '9'
  3261 = '= Setpoint'
  927 = 'A'
  753 = 'Absolute position used by "MOVE ABS"'
  519 = 'Action'
  149 = 'Action Legend:'
  6498 = 'Activate or deactivate early LN2 refilling'
  3985 = 'Activate or deactivate sensor heaters'
  849 = 'Activate sensor heater'
  5859 = 'Activates the Manual mode'
  1077 = 'Active'
  178 = 'Active Low'
  1017 = 'Actual Cmd'
  1932 = 'Actual command going out'
  2480 = 'Actual controller output'
  1403 = 'Actual Current'
  810 = 'Actual Duty Cycle'
  459 = 'Actual Input'
  3154 = 'Actual input temperature'
  1424 = 'Actual out'
  1070 = 'Actual Position'
  1863 = 'Actual Position [UU]'
  231 = 'Actual Power'
  545 = 'Actual Ramp'
  968 = 'Actual ramp value'
  123 = 'Actual Speed'
  405 = 'Actual Value'
  1303 = 'Actual Valve command '
  3192 = 'Actual variable setpoint temperature'
  795 = 'Additional information mostly used for description of errors'
  1764 = 'Alarm'
  4367 = 'Alarm Setpoint'
  202 = 'Ambiant'
  34 = 'Ambient Temperatures'
  936 = 'Anti-Fogging'
  531 = 'AUTO'
  2270 = 'Auto'
  1295 = 'AUTO Cmd'
  815 = 'Auto Disable'
  822 = 'Auto Disable Motor After Move'
  2792 = 'AUTO mode'
  1450 = 'Auto out'
  2697 = 'Automatic LN2 Filling'
  394 = 'Automatic LN2 Level Control'
  185 = 'Average'
  4108 = 'Average of all temperatures'
  3511 = 'Average Temp'
  938 = 'Axis Ready'
  171 = 'Axis Type'
  174 = 'Backlash'
  1705 = 'Beam Splitter'
  190 = 'Birefringence'
  4760 = 'Blower ON'
  964 = 'BLUE = Used\nBLANK = Not Used'
  3236 = 'Bottom'
  912 = 'Brake Active'
  507 = 'Brake Feedback Signal is Active Low'
  945 = 'Brake Used'
  173 = 'Brakes'
  177 = 'Brakes Used'
  716 = 'Branch A'
  1231 = 'Branch B'
  3748 = 'Busy'
  3965 = 'C'
  986 = 'Cabinets'
  2645 = 'Calculcated'
  3759 = 'Cause'
  837 = 'Cfg'
  1687 = 'CFO - Common Fore Optics'
  794 = 'Check'
  869 = 'Check the box if this is an SoE drive (Sercos over EtherCAT) , e.g. AX5000'
  176 = 'Cicular-Optimised'
  175 = 'Circular-Opt'
  960 = 'Clear diagnostics'
  836 = 'Clear NOVRAM'
  843 = 'Clear NOVRAM. Use it with care!\n\nThis is needed ONLY if NOVRAM was previously used for data structures different than T_MOTOR_CFG (or for previous versions of T_MOTOR_CFG).\nBring the motor to NOT_READY first and then clear NOVRAM.'
  1956 = 'CLOSE'
  4164 = 'Close Shutter'
  4466 = 'CO2 Pressure '
  5050 = 'CO2 Translation Stages'
  3040 = 'CO2 Translation StagesSplitter'
  226 = 'Cold'
  2331 = 'Comm errors'
  1799 = 'Command coming from the Control System'
  3843 = 'Compressor is running'
  523 = 'Compressor Year: '
  1260 = 'Config'
  206 = 'Continuously read all commands in the configuration'
  208 = 'Continuously read the User command'
  1589 = 'Control'
  1176 = 'Control Loops'
  877 = 'Control Units'
  932 = 'Controller Enabled'
  3499 = 'Controller Out'
  1406 = 'Controller State-Machine'
  3726 = 'Cool-Down'
  1365 = 'CoolDown'
  756 = 'Cooler Sleeves pressure Gauges'
  143 = 'Coolers'
  943 = 'Cooling Circuit pressure Gauges'
  485 = 'Cooling Down'
  1369 = 'CoolingDone'
  3960 = 'CRY - Cryostat'
  4373 = 'Cryo Interlocks'
  1011 = 'Cryo Temperatures'
  765 = 'Cryostat Pressures'
  989 = 'Current: '
  398 = 'D'
  6580 = 'Delay Lines'
  1575 = 'Delta Pressure\n%4.1f bar'
  3467 = 'Derivative action time'
  33 = 'Derivative part (Td)'
  475 = 'Detectors'
  862 = 'Dew point'
  1757 = 'Dew point calculation'
  763 = 'DISABLE'
  140 = 'Disable'
  1003 = 'DISABLE\nAXIS'
  1211 = 'Disable\nAxis'
  723 = 'Disable PID'
  335 = 'DL 1'
  889 = 'DL 2'
  831 = 'DL 3'
  126 = 'DL 4'
  1654 = 'Done'
  596 = 'During AUTO mode, continuously update the manual output'
  4866 = 'Early Refilling'
  1941 = 'Either shutter is opening or closing'
  866 = 'ENABLE'
  1208 = 'Enable'
  997 = 'ENABLE\nAXIS'
  833 = 'Enable\nAxis'
  867 = 'Enable Clear NOVRAM'
  7 = 'Enable control loop'
  275 = 'Enable PID'
  433 = 'Enabled'
  1445 = 'ENG'
  1572 = 'Engineering / Commissioning Mode'
  1132 = 'ENGINEERING MODE'
  55 = 'Error'
  1458 = 'Error Code: %d'
  856 = 'Evac Branch A'
  80 = 'Evac Branch B'
  211 = 'Evacuation'
  806 = 'Event'
  381 = 'Events'
  188 = 'First Valid'
  6194 = 'Fixed Configurations'
  404 = 'Fixed setpoint'
  881 = 'Fixed setpoint temperature'
  787 = 'Flag if motor is locked'
  2366 = 'Gain (Kp)'
  1216 = 'GBV'
  784 = 'GBV A'
  677 = 'GBV B'
  2231 = 'General settings'
  951 = 'GREEN = Enabled\nRED = Disabled'
  990 = 'GREEN = In Position\nBLANK = Not In Position (or not used)'
  925 = 'GREEN = Initialised\nRED = Not Initialised'
  958 = 'GREEN = Ready\nRED = Not Ready'
  2959 = 'Green if the input temperature is valid'
  2145 = 'Green if the variable setpoint temperature is valid'
  1560 = 'GREEN=Initialized\nRED=Not-initialized'
  1689 = 'Heater'
  3590 = 'Heater ON'
  2440 = 'Heater Open Loop'
  693 = 'Heater Short'
  3281 = 'Heater State'
  847 = 'Heaters'
  543 = 'Helium\n%4.1f ºC'
  2849 = 'High'
  476 = 'High '
  3628 = 'High Alam'
  86 = 'High Alarm'
  909 = 'High Pressure\n%4.1f bar'
  5731 = 'Highest of all temperatures'
  1483 = 'Highest Temp'
  184 = 'Highest Temperature'
  3529 = 'Home'
  3293 = 'Hours: '
  2488 = 'HPG'
  3302 = 'HPG1'
  263 = 'HPG2'
  855 = 'I '
  695 = 'ICS Interlocks'
  801 = "If active, check if the in-pos signal is active after the move completes. If it is not, it's a failure."
  2525 = 'If active, it is not safe to operate the motor.'
  808 = 'If checked, In-Position feedback signal is active low'
  628 = 'If ON, compressor is running'
  5 = 'If ON, compressor is simulated'
  1779 = 'If ON, ENG command is not safe!'
  640 = 'If ON, Heater circuit is open'
  339 = 'If ON, Heater is active'
  721 = 'If ON, Heater is in short circuit'
  879 = 'If ON, Heater is simulated.'
  681 = 'If ON, reading is in error.'
  195 = 'If ON, reading is in Warning'
  1304 = 'If ON, reading is valid.'
  2000 = 'If ON, there is an error in the SW implementation of permission handling.'
  182 = 'If ON, TMP pump is at its nominal speed, i.e. Ready.'
  561 = 'If ON, TMP pump is still spinning.'
  759 = 'If the motor is locked, during INIT the motor will not move and its position will be set to this value.'
  893 = 'IMG - Imager'
  3126 = 'In Good Vacuum'
  984 = 'In Position'
  829 = 'In-Pos Check'
  166 = 'INDEX'
  865 = 'INIT'
  162 = 'INIT Sequence Definition'
  516 = 'INIT sequence timeout in [ms].'
  971 = 'INIT Step'
  514 = 'INIT:'
  845 = 'Initialised'
  650 = 'Initialize'
  4814 = 'Initialized'
  1467 = 'Integral part (Tn)'
  282 = 'Interlock'
  915 = 'Intermediate'
  108 = 'KRDG? C'
  96 = 'KRDG? D'
  2420 = 'Lakeshore 336'
  853 = 'Laminar Setpoint'
  3970 = 'Last forced switch to MANUAL'
  4222 = 'Level Hold Time'
  168 = 'LHW'
  285 = 'LM-band Lakeshore 336'
  965 = 'LMS - LM-band Spectrograph'
  5737 = 'LN2 Absent Temp'
  234 = 'LN2 Detection Temp'
  1350 = 'LN2 detection temperature threshold'
  871 = 'LN2 level control'
  2943 = 'LN2 Level Control'
  3464 = 'LN2 Level Sensor'
  5538 = 'LN2 Levels Bottom Segment'
  4861 = 'LN2 Levels Intermediate Segment'
  246 = 'LN2 Levels Stiff Ring'
  3950 = 'LN2 Supply'
  482 = 'Load Configuration'
  812 = 'Local Control'
  752 = 'Lock'
  87 = 'Low'
  4958 = 'Low Alam'
  67 = 'Low Alarm'
  106 = 'Low Pressure\n%4.1f bar'
  3656 = 'Lowest of all temperatures'
  1181 = 'Lowest Temp'
  183 = 'Lowest Temperature'
  169 = 'LSTOP'
  98 = 'MANUAL'
  1446 = 'Manual'
  3475 = 'Manual Cmd'
  888 = 'MANUAL mode'
  306 = 'Manual Mode'
  2812 = 'Manual out'
  2947 = 'Manual output percentage'
  1042 = 'Manual Valve Control'
  705 = 'Manually start/Stop LN2 Level Control'
  1776 = 'Master Temp'
  142 = 'Maunal Out'
  1145 = 'Max cooldown rate'
  409 = 'Max Current'
  2619 = 'Max current:'
  298 = 'Max Power'
  2996 = 'Max power:'
  1898 = 'Max warming up rate'
  513 = 'Max:'
  1053 = 'Maximum time before the input temperature (and if used, the variable setpoint temperature) must be valid. Otherwise the Error flag is set, and the control mode is forced to MANUAL.'
  2573 = 'Maximum time that the input sensor can be invalid, before automatically switching to AUTO.'
  272 = 'Maximum time that the variable setpoint sensor can be invalid, before automatically switching to AUTO.'
  1089 = 'Measured'
  189 = 'Median'
  3110 = 'METIS Cryo Controller'
  58 = 'Middle'
  512 = 'Min:'
  105 = 'MONITOR'
  1486 = 'MONITOR USER'
  769 = 'MOVE ABS'
  355 = 'Move Absolute'
  610 = 'MOVE REL'
  1 = 'MOVE REL +'
  995 = 'MOVE REL -'
  1408 = 'Move Relative +'
  181 = 'Move Relative -'
  775 = 'MOVE VEL+'
  605 = 'MOVE VEL-'
  696 = 'Move Velocity +'
  1120 = 'Move Velocity -'
  515 = 'MOVE:'
  908 = 'N-band Lakeshore 336'
  910 = 'N2V 1'
  47 = 'N2V 2'
  1235 = 'NCP 1'
  1612 = 'NCP 2'
  2017 = 'NCP 3'
  3064 = 'NCP 4'
  3001 = 'NGP 1'
  426 = 'NGP 2'
  1090 = 'NGP 3'
  3319 = 'NGP 4'
  1653 = 'NOTT Instrument Control'
  6483 = 'NPC 1'
  6799 = 'NPC 2'
  3469 = 'NPC 3'
  6064 = 'NPC 4'
  4363 = 'NSH 1'
  4288 = 'NSH 2'
  488 = 'NSH 3'
  5927 = 'NSH 4'
  649 = 'NTPA 1'
  544 = 'NTPA 2'
  876 = 'NTPA 3'
  1943 = 'NTPA 4'
  289 = 'NTPB 1'
  832 = 'NTPB 2'
  26 = 'NTPB 3'
  153 = 'NTPB 4'
  324 = 'NTTA 1'
  36 = 'NTTA 2'
  704 = 'NTTA 3'
  423 = 'NTTA 4'
  564 = 'NTTB 1'
  739 = 'NTTB 2'
  351 = 'NTTB 3'
  597 = 'NTTB 4'
  3853 = 'OFF'
  1136 = 'Offset'
  1168 = 'Offset (REL)'
  2750 = 'Offset added to the setpoint (optional, put to 0 if not needed)'
  1524 = 'Oil\n%4.1f ºC'
  3510 = 'ON'
  212 = 'OPEN'
  6731 = 'Open Shutter'
  498 = 'Open-loop Motion'
  2683 = 'Operational'
  791 = 'Operational State'
  2784 = 'Output'
  595 = 'Output ramp'
  949 = 'P'
  2528 = 'Partial Vaccum'
  4088 = 'Partial Vacuum'
  4097 = 'Partially Cold'
  5638 = 'Partially OPEN'
  1437 = 'Permit CLOSE'
  803 = 'Permit OFF'
  93 = 'Permit ON'
  1308 = 'Permit OPEN'
  562 = 'PID in active mode'
  3524 = 'PID in Manual mode'
  1376 = 'Position (ABS)'
  113 = 'Position Control'
  510 = 'Position Difference'
  773 = 'Position:'
  509 = 'Positive, negative or zero (no backlash)'
  731 = 'POST-INIT'
  745 = 'POST-MOVE'
  732 = 'Power'
  148 = 'Power Outage'
  2018 = 'Power setpoint'
  4013 = 'Power supply error'
  914 = 'Powered'
  724 = 'PRE-INIT'
  738 = 'PRE-MOVE'
  2120 = 'Preconditions'
  814 = 'Pressure in mbar'
  526 = 'Pressures'
  4364 = 'Pressurized'
  283 = 'Pre_Cooling Valves'
  2454 = 'PTC #A'
  3383 = 'PTC #B'
  445 = 'PTC #C'
  758 = 'PTC 1'
  248 = 'PTC 2'
  413 = 'PTC 3'
  3133 = 'PTC-1 Running'
  1919 = 'PTC-2 Running'
  1139 = 'PTC-3 Running'
  358 = 'PTCs'
  4516 = 'Pulse Tube Cooler 1'
  4535 = 'Pulse Tube Cooler 2'
  370 = 'Pulse Tube Cooler 3'
  277 = 'Pulse Tube Year: '
  1038 = 'pump speed > 0 rpm'
  911 = 'Pumps'
  2643 = 'PVP A'
  2837 = 'PVP B'
  547 = 'PVV A1'
  576 = 'PVV A2'
  360 = 'PVV A3'
  764 = 'PVV A4'
  534 = 'PVV B1'
  737 = 'PVV B2'
  79 = 'PVV B3'
  676 = 'PVV B4'
  979 = 'PVV P1'
  187 = 'PVV P2'
  430 = 'PVV P3'
  1345 = 'PVV1'
  1079 = 'PVV2'
  1190 = 'PVV3'
  115 = 'PVV4'
  2805 = 'Ramp\ngenerator'
  627 = 'Ramp Down'
  555 = 'Ramp down limit'
  321 = 'Ramp Up'
  2050 = 'Ramp up limit'
  1834 = 'Ramp [K/min]'
  4828 = 'Re-Generation'
  838 = 'READ'
  197 = 'READ USER'
  4761 = 'Recovery: %s'
  919 = 'RED = Applied\nBLANK = Released'
  167 = 'REF'
  128 = 'Refilling Cycle Time'
  30 = 'Regeneration'
  3528 = 'Relative Humidity'
  207 = 'Relative Motion'
  2351 = 'Relative offset used by "MOVE REL"'
  21 = 'RESET'
  1520 = 'Reset'
  1568 = 'RESET Branch A Valves'
  1084 = 'RESET Branch B Valves'
  574 = 'RESET PVV_P Valves'
  1963 = 'RESET Venting Valves'
  2638 = 'Resistance:'
  3981 = 'RH measurement'
  3150 = 'RH sensor power command'
  2098 = 'RH sensor power status'
  977 = 'RPC Call Status'
  648 = 'S/N Compressor: '
  952 = 'S/N Panel:'
  754 = 'S/N Pulse Tube: '
  4561 = 'Safe to Start'
  6974 = 'Safe to Stop'
  501 = 'Save Configuration'
  709 = 'SCA - Single Conjugate Adaptive Optics'
  530 = 'Sensor input'
  3384 = 'Sensor input timeout'
  593 = 'Services'
  179 = 'Set'
  981 = 'Set point'
  615 = 'SET POS'
  1102 = 'Set Position'
  924 = 'Set Velocity [UU/s]'
  890 = 'Setpoint'
  3772 = 'Setpoint = controller output x scaling'
  2049 = 'Setpoint after the scaling was applied'
  2890 = 'Setpoint during alarm conditions'
  1644 = 'Setpoint offset'
  728 = 'Setpoint switch'
  371 = 'Setpoint to achieve laminar flow during normal operations. '
  511 = 'Setting both limits to 0 means that limits are not used.'
  969 = 'Shield A'
  2694 = 'Shield B'
  3200 = 'Shield C'
  939 = 'Shut ter1'
  528 = 'Shuter 1'
  742 = 'Shutter 1'
  858 = 'Shutter 2'
  344 = 'Shutter 3'
  618 = 'Shutter 4'
  5572 = 'Shutter Control'
  4392 = 'Shutter is closed'
  5273 = 'Shutter is Open'
  4060 = 'Shutter Speed'
  6591 = 'Shutter Speed (mm/sec)'
  549 = 'Shutter1'
  1660 = 'Shutters'
  4357 = 'Sim Ambiant Temp C'
  2568 = 'Sim Bottom H'
  5391 = 'Sim Bottom HA'
  623 = 'Sim Bottom L'
  4421 = 'Sim Bottom LA'
  5432 = 'Sim Cryostat Temp'
  2829 = 'Sim Dew Point Temp C'
  935 = 'Sim Highest Temp'
  6416 = 'Sim Intermediate H'
  3569 = 'Sim Intermediate HA'
  4256 = 'Sim Intermediate L'
  1213 = 'Sim Intermediate LA'
  4052 = 'Sim Lowest Temp'
  5656 = 'Sim Rad Shields Temp'
  5733 = 'Sim Stiff Ring H'
  5417 = 'Sim Stiff Ring HA'
  3362 = 'Sim Stiff Ring L'
  2937 = 'Sim Stiff Ring LA'
  3826 = 'Sim Window Mount Temp C'
  1346 = 'Simulated value [C] when simulation is active.'
  698 = 'Simulated value [K] when simulation is active.'
  1553 = 'Simulation'
  882 = 'Simulation:'
  1449 = 'Single read of all commands in the configuration'
  198 = 'Single read of user command'
  868 = 'SoE Drive'
  3448 = 'Sorption Pump'
  1704 = 'Sorption-Pump Temps'
  2051 = 'Source'
  6901 = 'Speed'
  1111 = 'Speed (Pos)'
  1135 = 'Speed (Vel)'
  19 = 'START'
  653 = 'Startup mode'
  8 = 'Startup timeout'
  227 = 'Stat'
  1059 = 'stat.lrArrReadings[0].lrValue'
  1055 = 'stat.lrArrReadings[1].lrValue'
  419 = 'stat.lrArrReadings[20].lrValue'
  926 = 'stat.lrArrReadings[21].lrValue'
  782 = 'State'
  850 = 'Status'
  800 = 'Status Description'
  1490 = 'Stiff Ring'
  10 = 'STOP'
  1035 = 'STOP MONITOR'
  1039 = 'Stop Monitoring if in OP/MONITORIN state.'
  788 = 'Substate'
  280 = 'Subsystems'
  172 = 'SW Limits'
  575 = 'Switch between the fixed and the variable setpoint'
  517 = 'Switch exit timeout in [ms].'
  1377 = 'Switch to AUTO Mode'
  1785 = 'Switch to MANUAL Mode'
  518 = 'SWITCH:'
  601 = 'Switches'
  163 = 'Switches \nActive Low'
  2451 = 'Sync to Auto out in Auto mode'
  2613 = 'System is ready for operations'
  2982 = 'System ON'
  1949 = 'System Temperatures'
  401 = 'T Control ramp values'
  1973 = 'T1 -X10'
  443 = 'T1 -X9'
  1137 = 'T2 -X10'
  1839 = 'T2 -X11'
  363 = 'T3 -X12'
  464 = 'Target'
  1119 = 'Target              Actual'
  1273 = 'Target ramp setpoint'
  2663 = 'Target setpoint'
  193 = 'Temp 1'
  319 = 'Temp 2'
  44 = 'Temp 3'
  210 = 'Temp 4'
  43 = 'Temp 5'
  59 = 'Temp Control'
  4099 = 'Temp thresholds for LN2 detection and temperature hysteresis'
  4138 = 'Temperature Control Loops'
  286 = 'Temperature in C'
  1950 = 'Temperature Thresholds'
  111 = 'Temperatures'
  5013 = 'Temporal Hysteresis'
  766 = 'The motor will not move, if the target position is closer to the locked position than this value.'
  4563 = 'These configurations are used when no PID control is available.'
  6663 = 'Tilt A'
  1427 = 'Tilt B'
  1065 = 'Time to hold a change of status to avoid transient oscillations. '
  2407 = 'Time:'
  170 = 'Timeouts [ms]'
  3386 = 'Tip A'
  1236 = 'Tip B'
  1343 = 'Tip Tilt'
  1909 = 'TMP A'
  4137 = 'TMP B'
  1773 = 'Toggle Engineering Mode'
  780 = 'Tolerance:'
  1268 = 'Total Duration'
  4810 = 'TP Coolant Valves'
  487 = 'TPC A'
  3187 = 'TPC B'
  2386 = 'Transient ramp setpoint'
  165 = 'UHW'
  1948 = 'Unsafe!'
  717 = 'User \nProcs'
  2343 = 'User description'
  1009 = "User Units: '%s'"
  164 = 'USTOP'
  439 = 'UTC Time'
  1363 = 'Vacuum Achieved'
  996 = 'Vacuum pressure Gauges'
  253 = 'VAGA1'
  146 = 'VAGA2'
  970 = 'VAGA3'
  1502 = 'VAGB1'
  682 = 'VAGB2'
  120 = 'VAGB3'
  455 = 'VAGF'
  1488 = 'VAGF1'
  1083 = 'VAGF2'
  2485 = 'VAGG'
  620 = 'VAGG1'
  1498 = 'VAGG2'
  743 = 'Valid'
  180 = 'Value 1'
  345 = 'Value 2'
  1854 = 'Value used by the system [C]'
  1212 = 'Value used by the system [K]'
  4193 = 'Valve Cmd'
  408 = 'Valve ctrl'
  473 = 'Valve Open'
  616 = 'Valve open (0 - 100)%'
  973 = 'Valve State'
  1494 = 'Valve state: ON=OPEN, OFF=CLOSED'
  1423 = 'Valves'
  2175 = 'Variable setpoint'
  425 = 'Variable setpoint timeout'
  1373 = 'Vent'
  270 = 'Venting'
  826 = 'Venting Valves'
  1112 = 'VentingDone'
  1016 = 'Ver: %s'
  1634 = 'vote Temperature'
  4186 = 'Voter outputs'
  3715 = 'Voters'
  524 = 'Voting Temperature out [K]'
  726 = 'W'
  3991 = 'Warm'
  3798 = 'Warm Pressurized'
  1360 = 'Warm Vacuum'
  1618 = 'Warm-Up'
  2893 = 'Warming Up'
  448 = 'WarmUp'
  1380 = 'WarmUpDone'
  672 = 'Warning'
  14 = 'Warning High Sensor'
  873 = 'Warning High-Alarm Sensor'
  1319 = 'Warning Low Sensor'
  354 = 'Warning Low-Alarm Sensor'
  918 = 'Water IN\n%4.1f ºC'
  57 = 'Water OUT\n%4.1f ºC'
  2737 = 'Window'
  2819 = 'x Scaling'
  4065 = 'ZnSe Actuators'
END_TEXTLIST

// ---- HMI/VISUs/Events/VISU_HMI_EVENTS.TcVIS
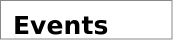
VISUALIZATION VISU_HMI_EVENTS  // 173x40
    Label (10,10 163x30), "Events"
END_VISUALIZATION

// ---- HMI/VISUs/Home/VISU_HMI_HOME.TcVIS
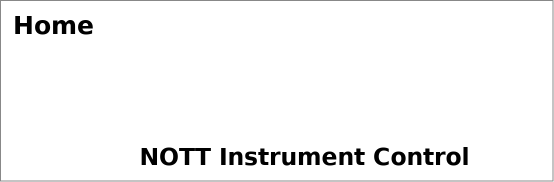
VISUALIZATION VISU_HMI_HOME  // 554x182
VAR_IN_OUT
	m_instance : FB_NOTT_ICS;
END_VAR
    Label (10,10 150x30), "Home"
    Label (56,132 498x50), "NOTT Instrument Control"
END_VISUALIZATION

// ---- HMI/VISUs/ICS_Interlocks/VISU_HMI_CRYO_INTERLOCKS.TcVIS
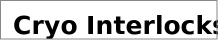
VISUALIZATION VISU_HMI_CRYO_INTERLOCKS  // 218x40
    Label (10,10 208x30), "Cryo Interlocks"
END_VISUALIZATION

// ---- HMI/VISUs/Services/VISU_HMI_SERVICES.TcVIS
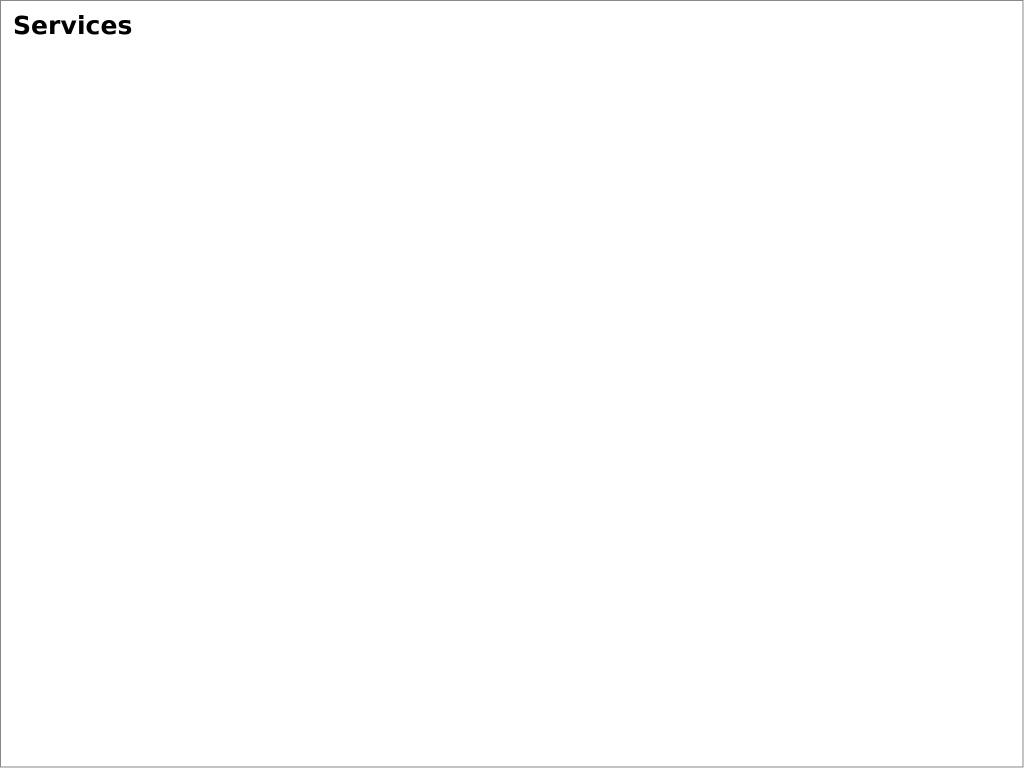
VISUALIZATION VISU_HMI_SERVICES  // 1024x768
VAR_IN_OUT
	m_Instance : FB_SERVICES;
    //m_Hmi : FB_HMI_SERVICES;
END_VAR
    Label (10,10 150x30), "Services"
END_VISUALIZATION

// ---- HMI/VISUs/Services/VISU_HMI_SERVICES_TIME.TcVIS
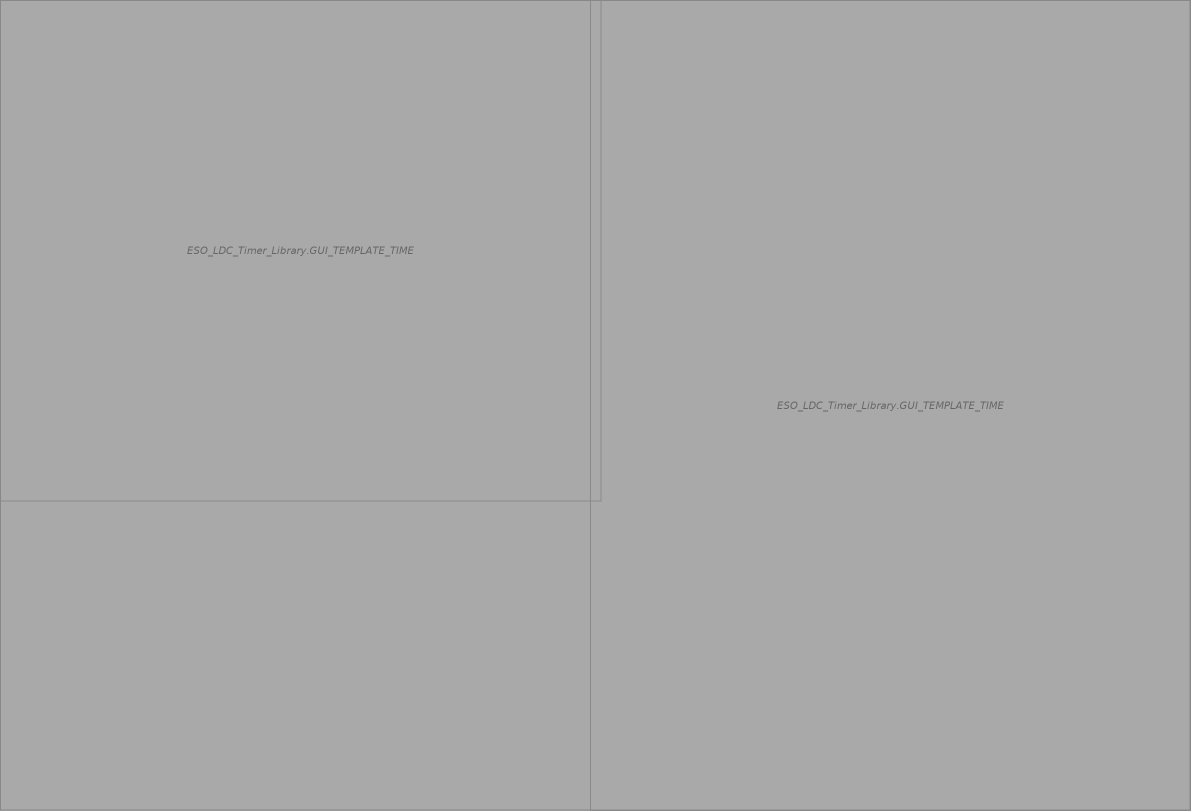
VISUALIZATION VISU_HMI_SERVICES_TIME  // 1191x811
VAR_IN_OUT
	m_Instance : FB_TIME;
    m_Hmi : FB_HMI_SERVICES_TIME;
END_VAR
    Frame (0,0 601x501)
        shows ESO_LDC_Timer_Library.GUI_TEMPLATE_TIME(m_DeviceName := 'time_info', m_Instance := m_Instance)
    Frame (590,0 601x811)
        shows ESO_LDC_Timer_Library.GUI_TEMPLATE_TIME(m_DeviceName := 'time_info', m_Instance := m_Instance)
        p2738717112: m_Hmi.nAbsoluteMovementY
END_VISUALIZATION

// ---- HMI/VISUs/Subsystems/Beam_Splitter/VISU_HMI_BEAM_SPLITTER.TcVIS
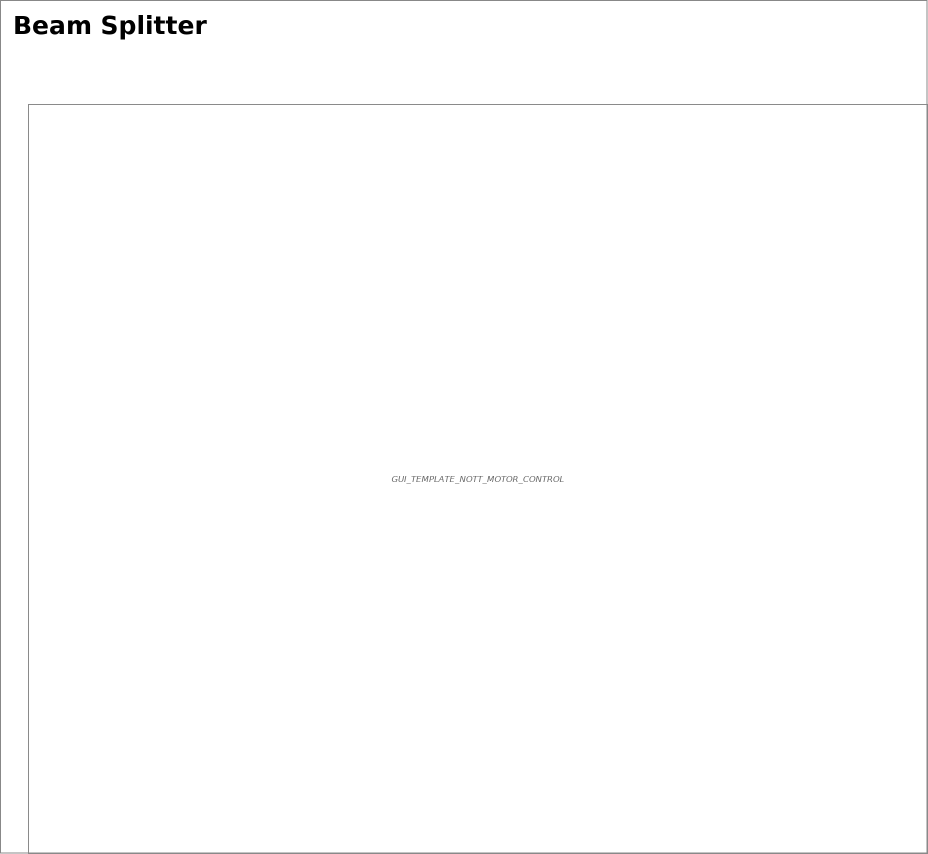
VISUALIZATION VISU_HMI_BEAM_SPLITTER  // 928x854
    Label (10,10 199x30), "Beam Splitter"
    Frame (28,104 900x750)
        shows GUI_TEMPLATE_MOTOR(m_Instance := MAIN.nott_ics.Calibration_Unit_Beam_Splitter.NBS)
END_VISUALIZATION

// ---- HMI/VISUs/Subsystems/Birefringence/VISU_HMI_BIREFRINGENCE.TcVIS
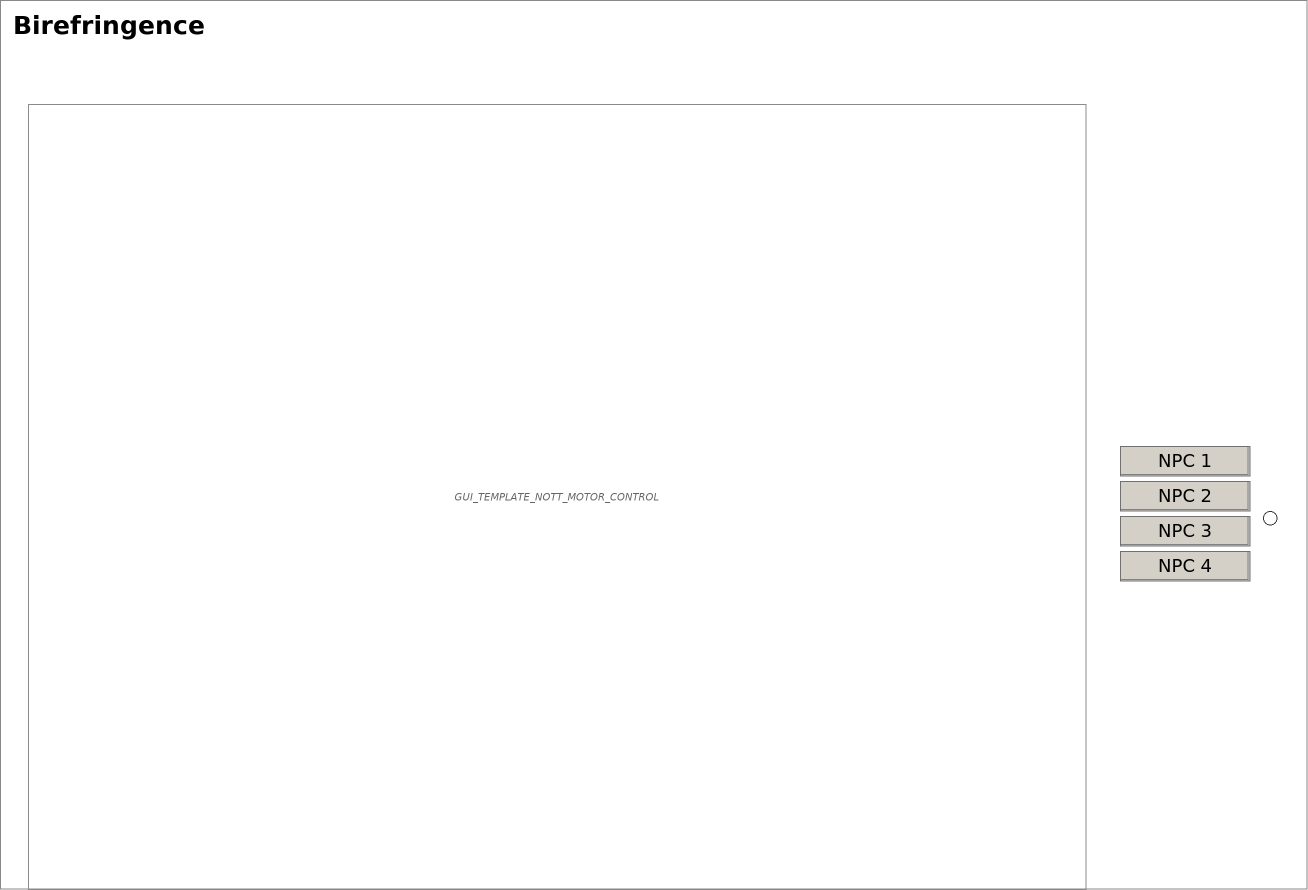
VISUALIZATION VISU_HMI_BIREFRINGENCE  // 1308x890
    Label (10,10 199x30), "Birefringence"
    Frame (28,104 1058x786)
        shows GUI_TEMPLATE_MOTOR(m_Instance := MAIN.nott_ics.Birefringence.ptrNPCs[MAIN.nott_ics.Birefringence.guiNPCsIndex]^)
    RadioButton (1261,448 47x140), variable: MAIN.nott_ics.Birefringence.guiNPCsIndex-1
        Areas[0]: Text=Radiobutton
        Areas[1]: Text=Radiobutton
    Button (1120,446 130x30), "NPC 1"
        OnMouseClick: execute { MAIN.nott_ics.Birefringence.guiNPCsIndex := 1; }
    Button (1120,481 130x30), "NPC 2"
        OnMouseClick: execute { MAIN.nott_ics.Birefringence.guiNPCsIndex := 2; }
    Button (1120,516 130x30), "NPC 3"
        OnMouseClick: execute { MAIN.nott_ics.Birefringence.guiNPCsIndex := 3; }
    Button (1120,551 130x30), "NPC 4"
        OnMouseClick: execute { MAIN.nott_ics.Birefringence.guiNPCsIndex := 4; }
END_VISUALIZATION

// ---- HMI/VISUs/Subsystems/CO2_Pressure/VISU_HMI_CO2_PRESSURE.TcVIS
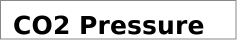
VISUALIZATION VISU_HMI_CO2_PRESSURE  // 237x40
    Label (10,10 227x30), "CO2 Pressure"
END_VISUALIZATION

// ---- HMI/VISUs/Subsystems/CO2_Translation_Stages/VISU_HMI_CO2_TRANS_STAGES.TcVIS
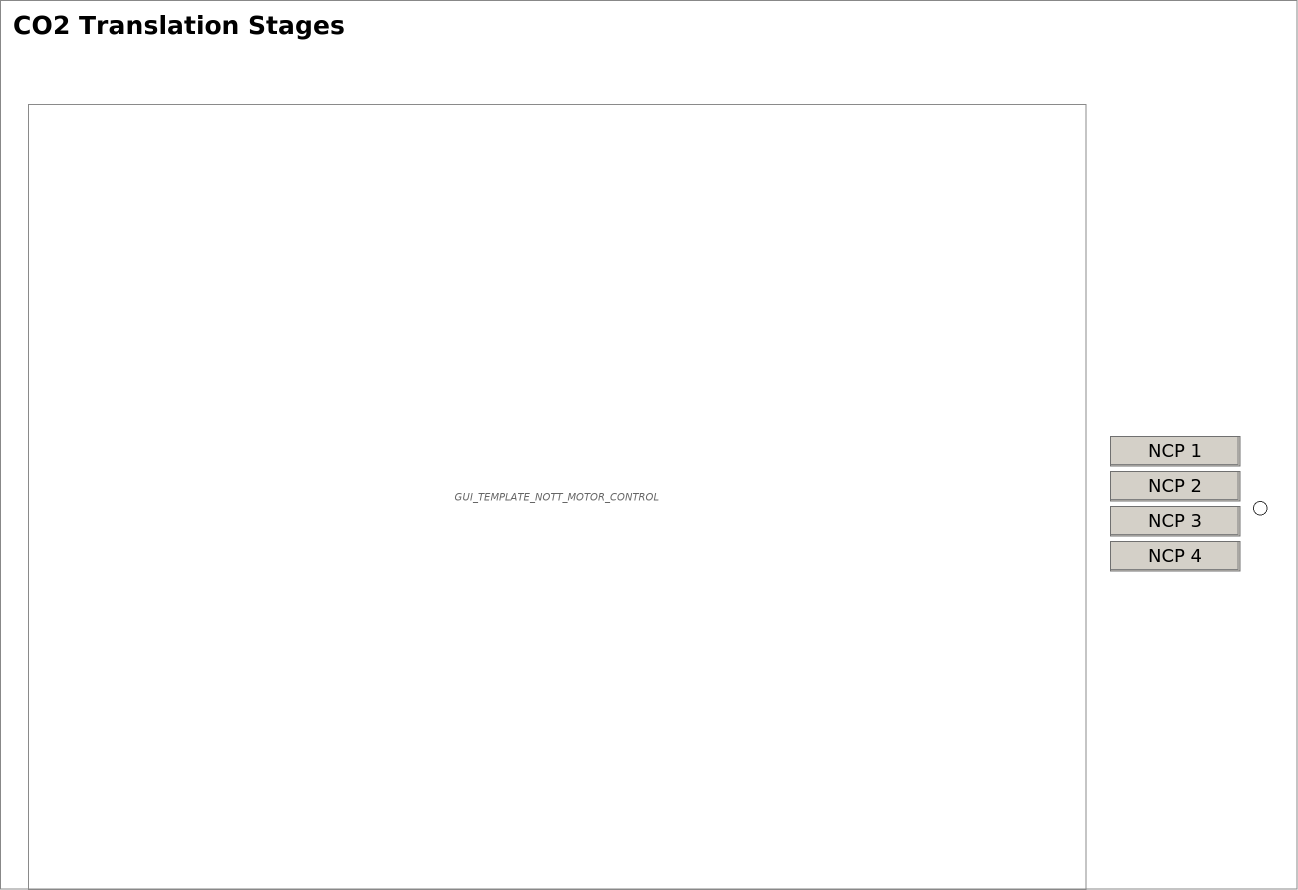
VISUALIZATION VISU_HMI_CO2_TRANS_STAGES  // 1298x890
    Label (10,10 379x30), "CO2 Translation Stages"
    Frame (28,104 1058x786)
        shows GUI_TEMPLATE_MOTOR(m_Instance := MAIN.nott_ics.CO2TransStages.ptrNCPs[MAIN.nott_ics.CO2TransStages.guiNCPsIndex]^)
    RadioButton (1251,438 47x140), variable: MAIN.nott_ics.CO2TransStages.guiNCPsIndex-1
        Areas[0]: Text=Radiobutton
        Areas[1]: Text=Radiobutton
    Button (1110,436 130x30), "NCP 1"
        OnMouseClick: execute { MAIN.nott_ics.CO2TransStages.guiNCPsIndex := 1; }
    Button (1110,471 130x30), "NCP 2"
        OnMouseClick: execute { MAIN.nott_ics.CO2TransStages.guiNCPsIndex := 2; }
    Button (1110,506 130x30), "NCP 3"
        OnMouseClick: execute { MAIN.nott_ics.CO2TransStages.guiNCPsIndex := 3; }
    Button (1110,541 130x30), "NCP 4"
        OnMouseClick: execute { MAIN.nott_ics.CO2TransStages.guiNCPsIndex := 4; }
END_VISUALIZATION

// ---- HMI/VISUs/Subsystems/DelayLines/VISU_HMI_DELAY_LINES.TcVIS
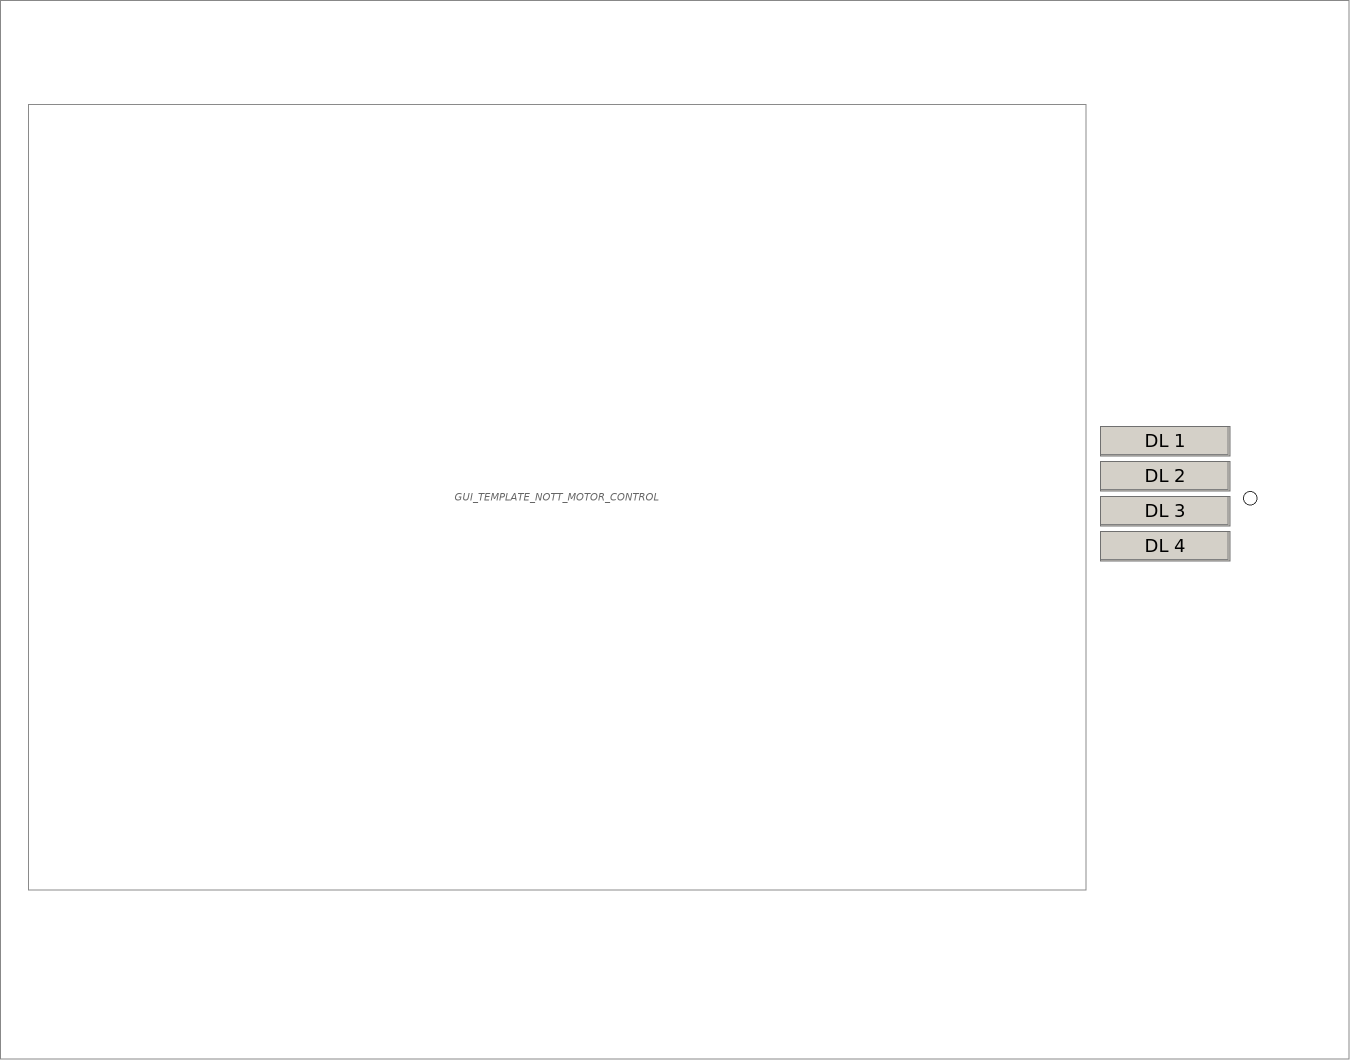
VISUALIZATION VISU_HMI_DELAY_LINES  // 1350x1060
    Label (10,10 199x30), "Delay Lines"
    Frame (28,104 1058x786)
        shows GUI_TEMPLATE_MOTOR(m_Instance := MAIN.nott_ics.Delay_Lines.ptrDelayLines[MAIN.nott_ics.Delay_Lines.guiDLIndex]^)
    RadioButton (1241,428 47x140), variable: MAIN.nott_ics.Delay_Lines.guiDLIndex-1
        Areas[0]: Text=Radiobutton
        Areas[1]: Text=Radiobutton
    Button (1100,426 130x30), "DL 1"
        OnMouseClick: execute { MAIN.nott_ics.Delay_Lines.guiDLIndex := 1; }
    Button (1100,461 130x30), "DL 2"
        OnMouseClick: execute { MAIN.nott_ics.Delay_Lines.guiDLIndex := 2; }
    Button (1100,496 130x30), "DL 3"
        OnMouseClick: execute { MAIN.nott_ics.Delay_Lines.guiDLIndex := 3; }
    Button (1100,531 130x30), "DL 4"
        OnMouseClick: execute { MAIN.nott_ics.Delay_Lines.guiDLIndex := 4; }
END_VISUALIZATION

// ---- HMI/VISUs/Subsystems/Shutters/VISU_HMI_SHUTTERS.TcVIS
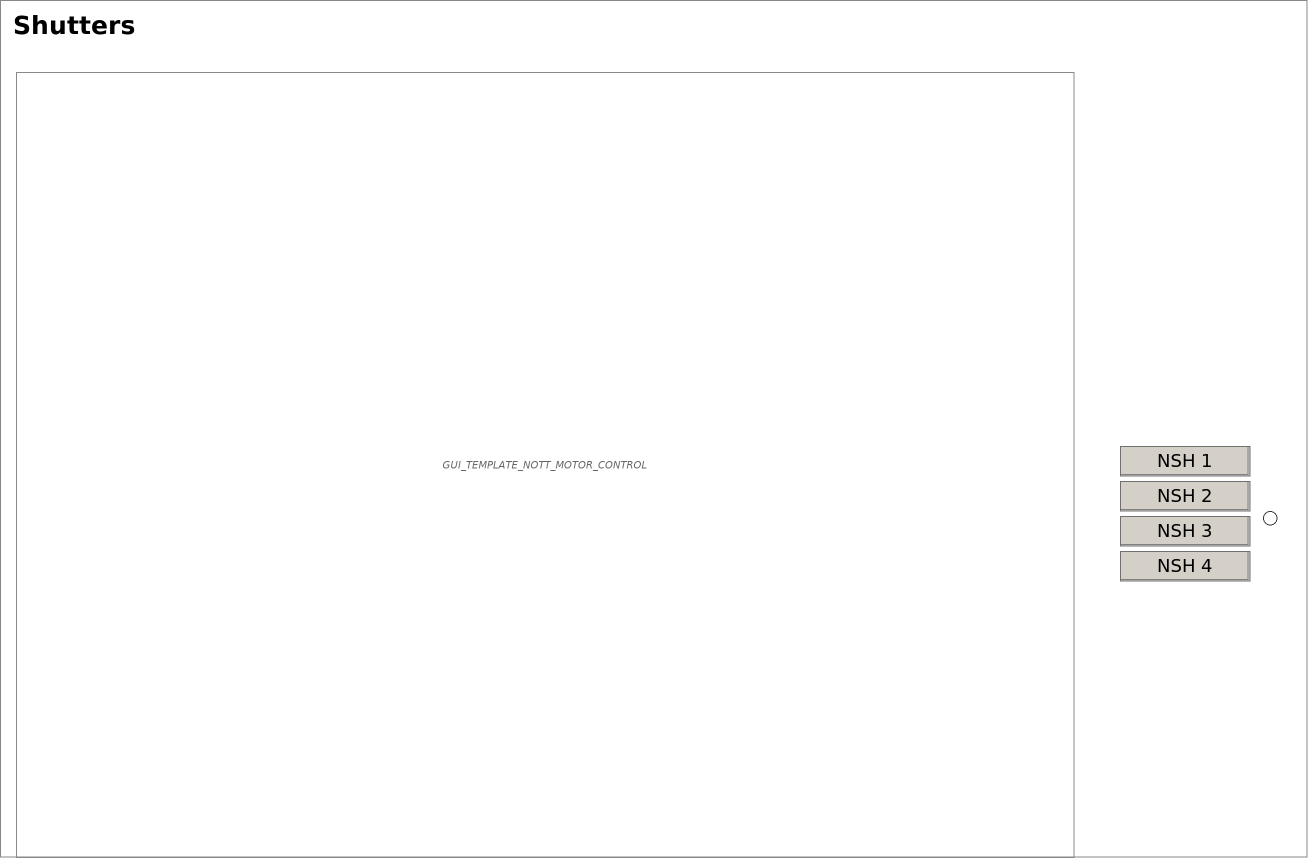
VISUALIZATION VISU_HMI_SHUTTERS  // 1308x858
    Label (10,10 199x30), "Shutters"
    RadioButton (1261,448 47x140), variable: MAIN.nott_ics.Shutters.guiShutterIndex-1
        Areas[0]: Text=Radiobutton
        Areas[1]: Text=Radiobutton
    Button (1120,446 130x30), "NSH 1"
        OnMouseClick: execute { MAIN.nott_ics.Shutters.guiShutterIndex := 1; }
    Button (1120,481 130x30), "NSH 2"
        OnMouseClick: execute { MAIN.nott_ics.Shutters.guiShutterIndex := 2; }
    Button (1120,516 130x30), "NSH 3"
        OnMouseClick: execute { MAIN.nott_ics.Shutters.guiShutterIndex := 3; }
    Button (1120,551 130x30), "NSH 4"
        OnMouseClick: execute { MAIN.nott_ics.Shutters.guiShutterIndex := 4; }
    Frame (16,72 1058x786)
        shows GUI_TEMPLATE_MOTOR(m_Instance := MAIN.nott_ics.Shutters.ptrShutters[MAIN.nott_ics.Shutters.guiShutterIndex]^)
END_VISUALIZATION

// ---- HMI/VISUs/Subsystems/TipTilt/Components/VISU_HMI_TILT_A.TcVIS
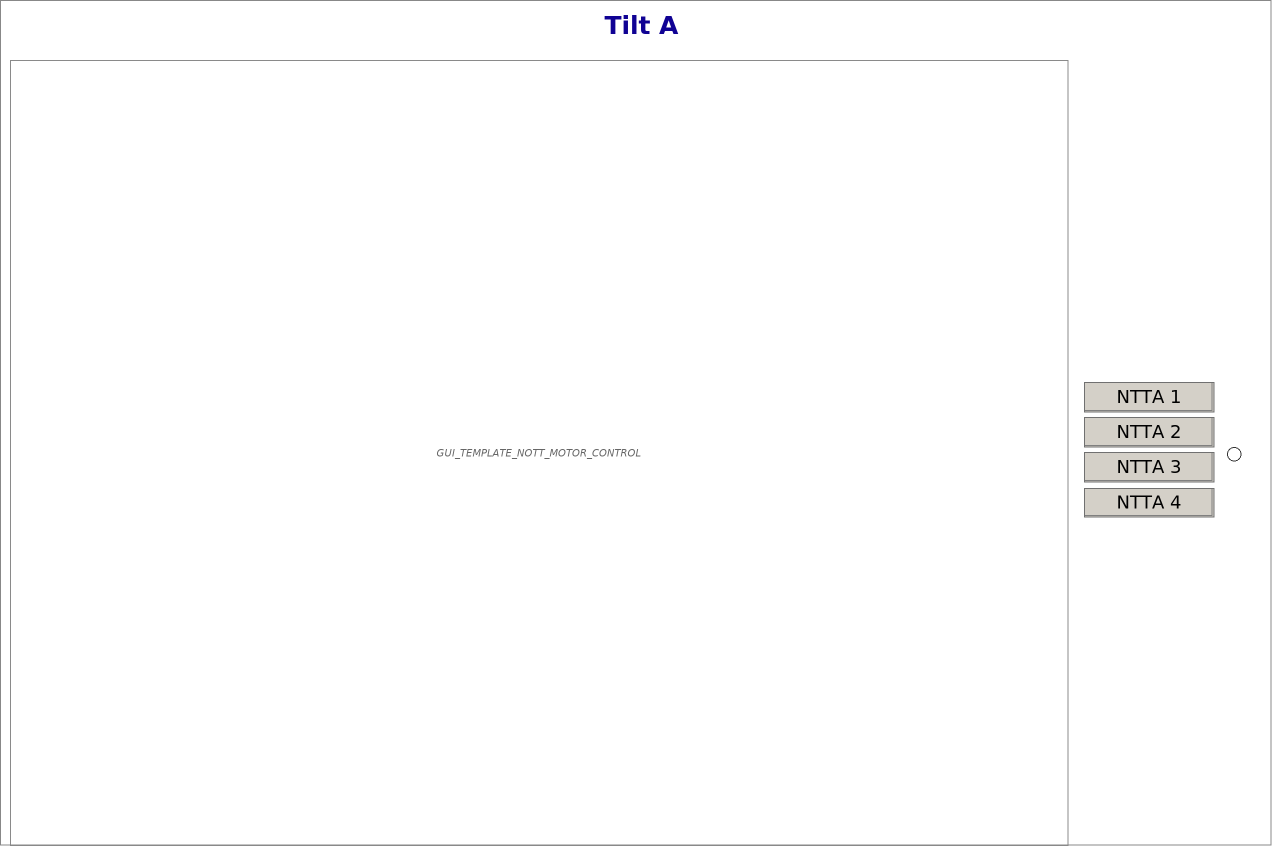
VISUALIZATION VISU_HMI_TILT_A  // 1272x846
    Group (10,60 1262x786)
        Frame (0,0 1058x786)
            shows GUI_TEMPLATE_MOTOR(m_Instance := MAIN.nott_ics.TipTilt.ptrTiltActuatorsA[MAIN.nott_ics.TipTilt.guiTiltActuatorsAIndex]^)
        Group (1074,322 188x142)
            RadioButton (141,2 47x140), variable: MAIN.nott_ics.TipTilt.guiTiltActuatorsAIndex-1
                Areas[0]: Text=Radiobutton
                Areas[1]: Text=Radiobutton
            Button (0,0 130x30), "NTTA 1"
                OnMouseClick: execute { MAIN.nott_ics.TipTilt.guiTiltActuatorsAIndex := 1; }
            Button (0,35 130x30), "NTTA 2"
                OnMouseClick: execute { MAIN.nott_ics.TipTilt.guiTiltActuatorsAIndex := 2; }
            Button (0,70 130x30), "NTTA 3"
                OnMouseClick: execute { MAIN.nott_ics.TipTilt.guiTiltActuatorsAIndex := 3; }
            Button (0,106 130x29), "NTTA 4"
                OnMouseClick: execute { MAIN.nott_ics.TipTilt.guiTiltActuatorsAIndex := 4; }
    Label (542,10 199x30), "Tilt A"
END_VISUALIZATION

// ---- HMI/VISUs/Subsystems/TipTilt/Components/VISU_HMI_TILT_B.TcVIS
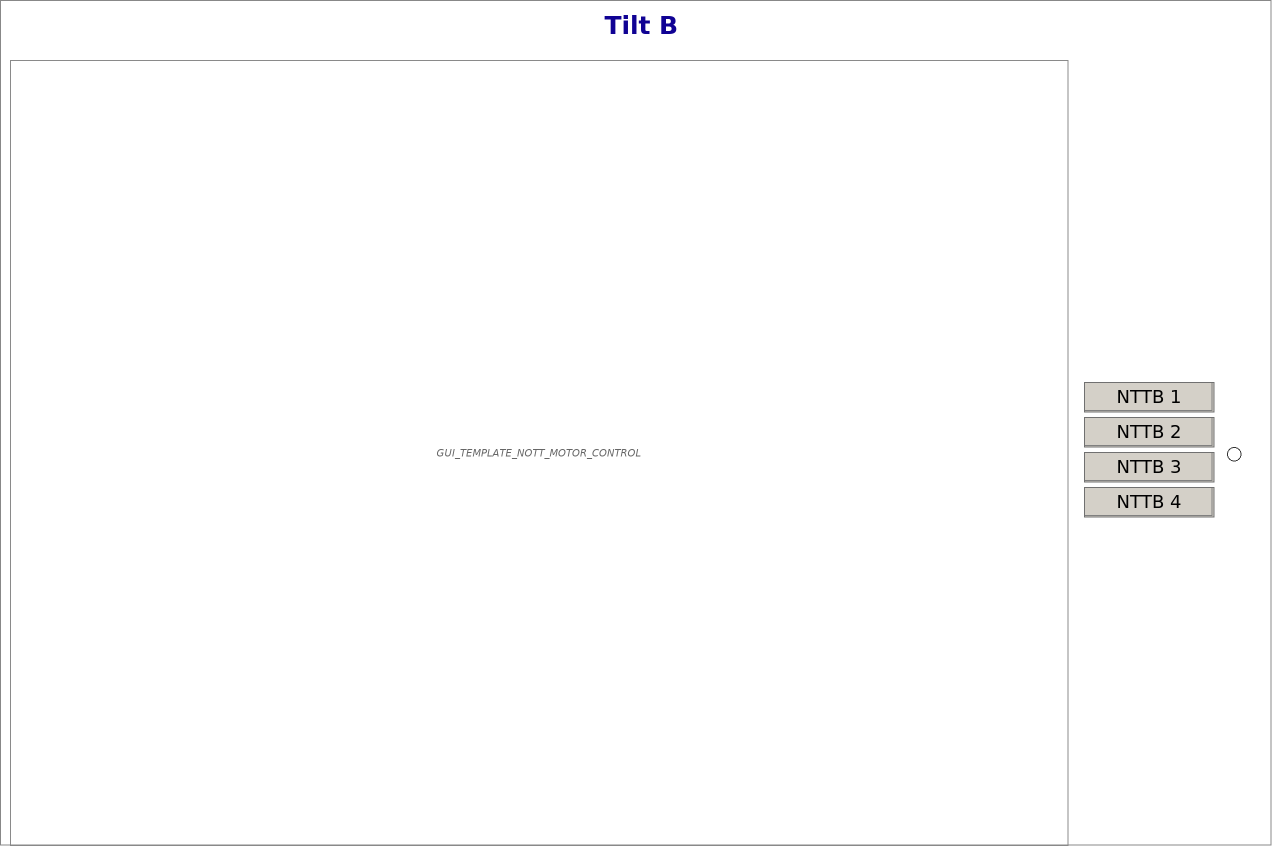
VISUALIZATION VISU_HMI_TILT_B  // 1272x846
    Label (542,10 199x30), "Tilt B"
    Group (10,60 1262x786)
        Frame (0,0 1058x786)
            shows GUI_TEMPLATE_MOTOR(m_Instance := MAIN.nott_ics.TipTilt.ptrTiltActuatorsB[MAIN.nott_ics.TipTilt.guiTiltActuatorsBIndex]^)
        Group (1074,322 188x142)
            RadioButton (141,2 47x140), variable: MAIN.nott_ics.TipTilt.guiTiltActuatorsBIndex-1
                Areas[0]: Text=Radiobutton
                Areas[1]: Text=Radiobutton
            Button (0,0 130x30), "NTTB 1"
                OnMouseClick: execute { MAIN.nott_ics.TipTilt.guiTiltActuatorsBIndex := 1; }
            Button (0,35 130x30), "NTTB 2"
                OnMouseClick: execute { MAIN.nott_ics.TipTilt.guiTiltActuatorsBIndex := 2; }
            Button (0,70 130x30), "NTTB 3"
                OnMouseClick: execute { MAIN.nott_ics.TipTilt.guiTiltActuatorsBIndex := 3; }
            Button (0,105 130x30), "NTTB 4"
                OnMouseClick: execute { MAIN.nott_ics.TipTilt.guiTiltActuatorsBIndex := 4; }
END_VISUALIZATION

// ---- HMI/VISUs/Subsystems/TipTilt/Components/VISU_HMI_TIP_A.TcVIS
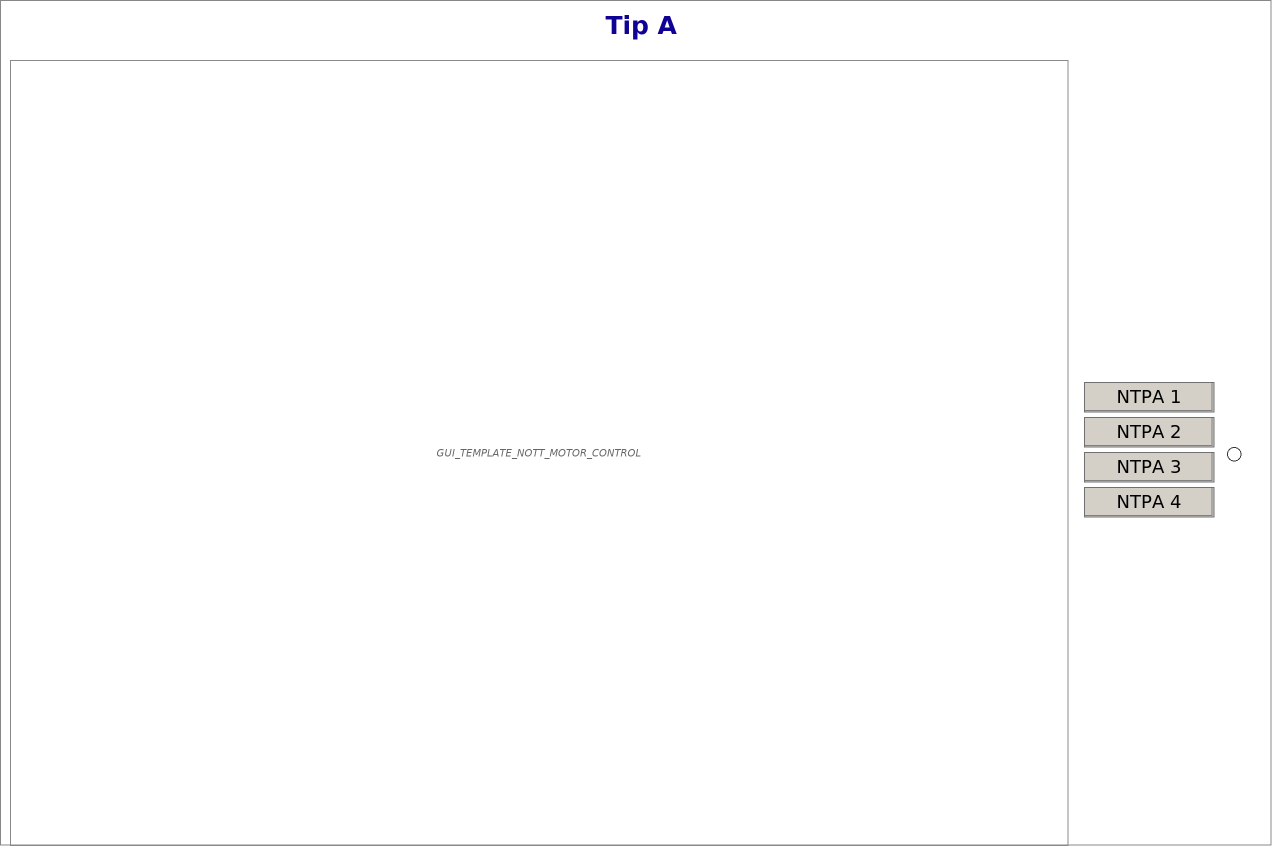
VISUALIZATION VISU_HMI_TIP_A  // 1272x846
    Group (10,10 1262x836)
        Label (532,0 199x30), "Tip A"
        Frame (0,50 1058x786)
            shows GUI_TEMPLATE_MOTOR(m_Instance := MAIN.nott_ics.TipTilt.ptrTipActuatorsA[MAIN.nott_ics.TipTilt.guiTipActuatorsAIndex]^)
        RadioButton (1215,374 47x140), variable: MAIN.nott_ics.TipTilt.guiTipActuatorsAIndex-1
            Areas[0]: Text=Radiobutton
            Areas[1]: Text=Radiobutton
        Button (1074,372 130x30), "NTPA 1"
            OnMouseClick: execute { MAIN.nott_ics.TipTilt.guiTipActuatorsAIndex := 1; }
        Button (1074,407 130x30), "NTPA 2"
            OnMouseClick: execute { MAIN.nott_ics.TipTilt.guiTipActuatorsAIndex := 2; }
        Button (1074,442 130x30), "NTPA 3"
            OnMouseClick: execute { MAIN.nott_ics.TipTilt.guiTipActuatorsAIndex := 3; }
        Button (1074,477 130x30), "NTPA 4"
            OnMouseClick: execute { MAIN.nott_ics.TipTilt.guiTipActuatorsAIndex := 4; }
END_VISUALIZATION

// ---- HMI/VISUs/Subsystems/TipTilt/Components/VISU_HMI_TIP_B.TcVIS
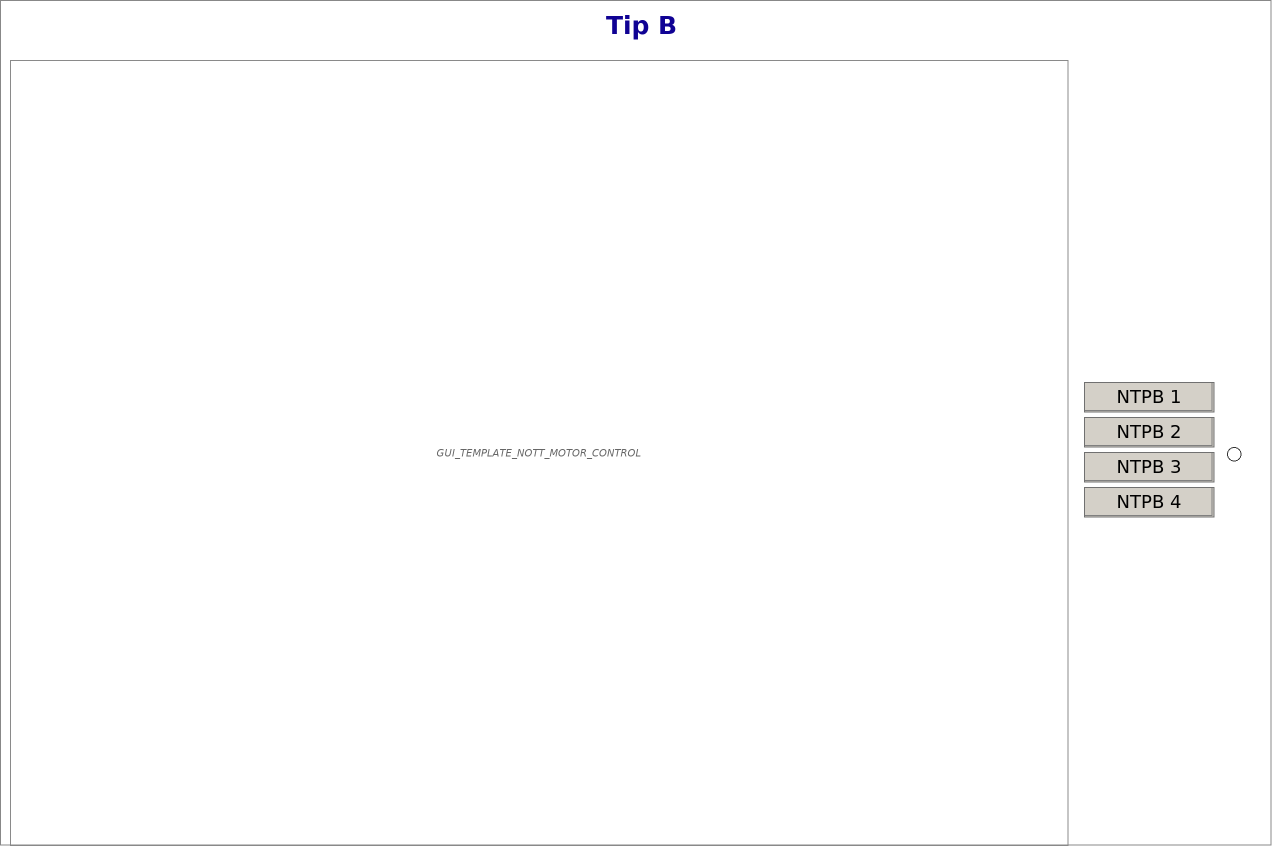
VISUALIZATION VISU_HMI_TIP_B  // 1272x846
    Label (542,10 199x30), "Tip B"
    Group (10,60 1262x786)
        Frame (0,0 1058x786)
            shows GUI_TEMPLATE_MOTOR(m_Instance := MAIN.nott_ics.TipTilt.ptrTipActuatorsB[MAIN.nott_ics.TipTilt.guiTipActuatorsBIndex]^)
        Group (1074,322 188x142)
            RadioButton (141,2 47x140), variable: MAIN.nott_ics.TipTilt.guiTipActuatorsBIndex-1
                Areas[0]: Text=Radiobutton
                Areas[1]: Text=Radiobutton
            Button (0,0 130x30), "NTPB 1"
                OnMouseClick: execute { MAIN.nott_ics.TipTilt.guiTipActuatorsBIndex := 1; }
            Button (0,35 130x30), "NTPB 2"
                OnMouseClick: execute { MAIN.nott_ics.TipTilt.guiTipActuatorsBIndex := 2; }
            Button (0,70 130x30), "NTPB 3"
                OnMouseClick: execute { MAIN.nott_ics.TipTilt.guiTipActuatorsBIndex := 3; }
            Button (0,105 130x30), "NTPB 4"
                OnMouseClick: execute { MAIN.nott_ics.TipTilt.guiTipActuatorsBIndex := 4; }
END_VISUALIZATION

// ---- HMI/VISUs/Subsystems/TipTilt/VISU_HMI_TIP_TILT.TcVIS
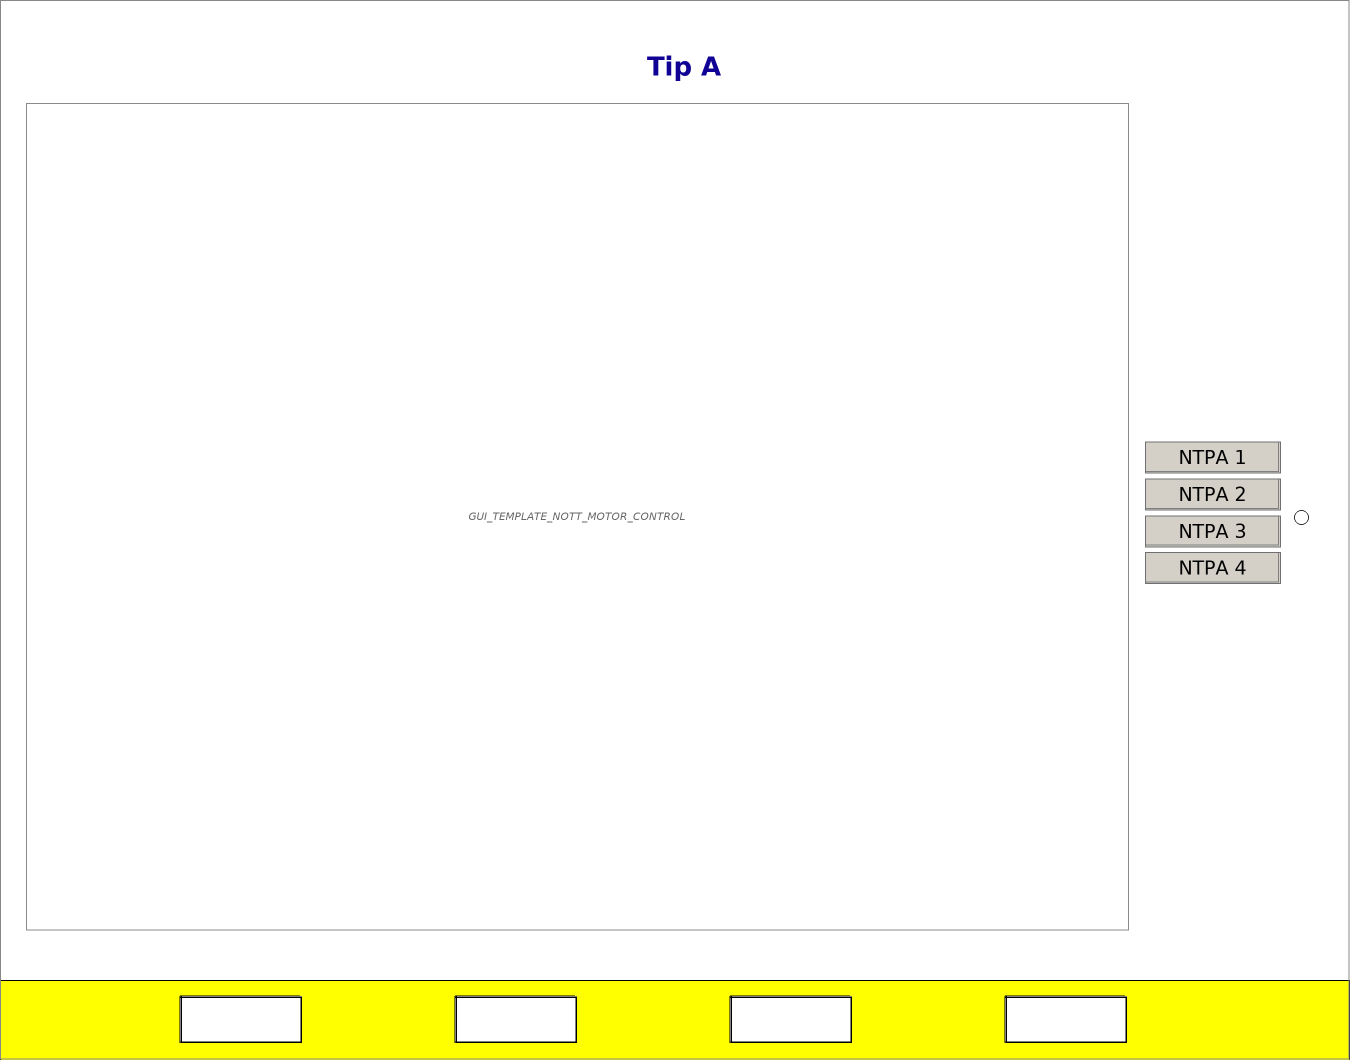
VISUALIZATION VISU_HMI_TIP_TILT  // 1350x1060
VAR_IN_OUT
	m_Hmi : FB_HMI_TIP_TILT;
END_VAR
    Label (10,10 199x30), "Tip Tilt"
    Rectangle (0,980 1350x81)
    Frame (180,996 123x48)
        shows VISU_HMI_SUBSYSTEM_BUTTON(m_Hmi := PRG_HMI.fbTipTilt.fbTipAButton)
        OnMouseClick: execute { m_Hmi.eActiveTab := E_HMI_TIP_TILT_TABS.TIP_A; }
    Frame (455,996 123x48)
        shows VISU_HMI_SUBSYSTEM_BUTTON(m_Hmi := PRG_HMI.fbTipTilt.fbTipBButton)
        OnMouseClick: execute { m_Hmi.eActiveTab := E_HMI_TIP_TILT_TABS.TIP_B; }
    Frame (730,996 123x48)
        shows VISU_HMI_SUBSYSTEM_BUTTON(m_Hmi := PRG_HMI.fbTipTilt.fbTiltAButton)
        OnMouseClick: execute { m_Hmi.eActiveTab := E_HMI_TIP_TILT_TABS.TILT_A; }
    Frame (1005,996 123x48)
        shows VISU_HMI_SUBSYSTEM_BUTTON(m_Hmi := PRG_HMI.fbTipTilt.fbTiltBButton)
        OnMouseClick: execute { m_Hmi.eActiveTab := E_HMI_TIP_TILT_TABS.TILT_B; }
    Frame (16,40 1325x890), frame switch variable: m_Hmi.eActiveTab
        shows VISU_HMI_TIP_A()
        shows VISU_HMI_TIP_B()
        shows VISU_HMI_TILT_A()
        shows VISU_HMI_TILT_B()
END_VISUALIZATION

// ---- HMI/VISUs/Subsystems/ZnSe_Actuators/VISU_HMI_ZNSE_ACTUATORS.TcVIS
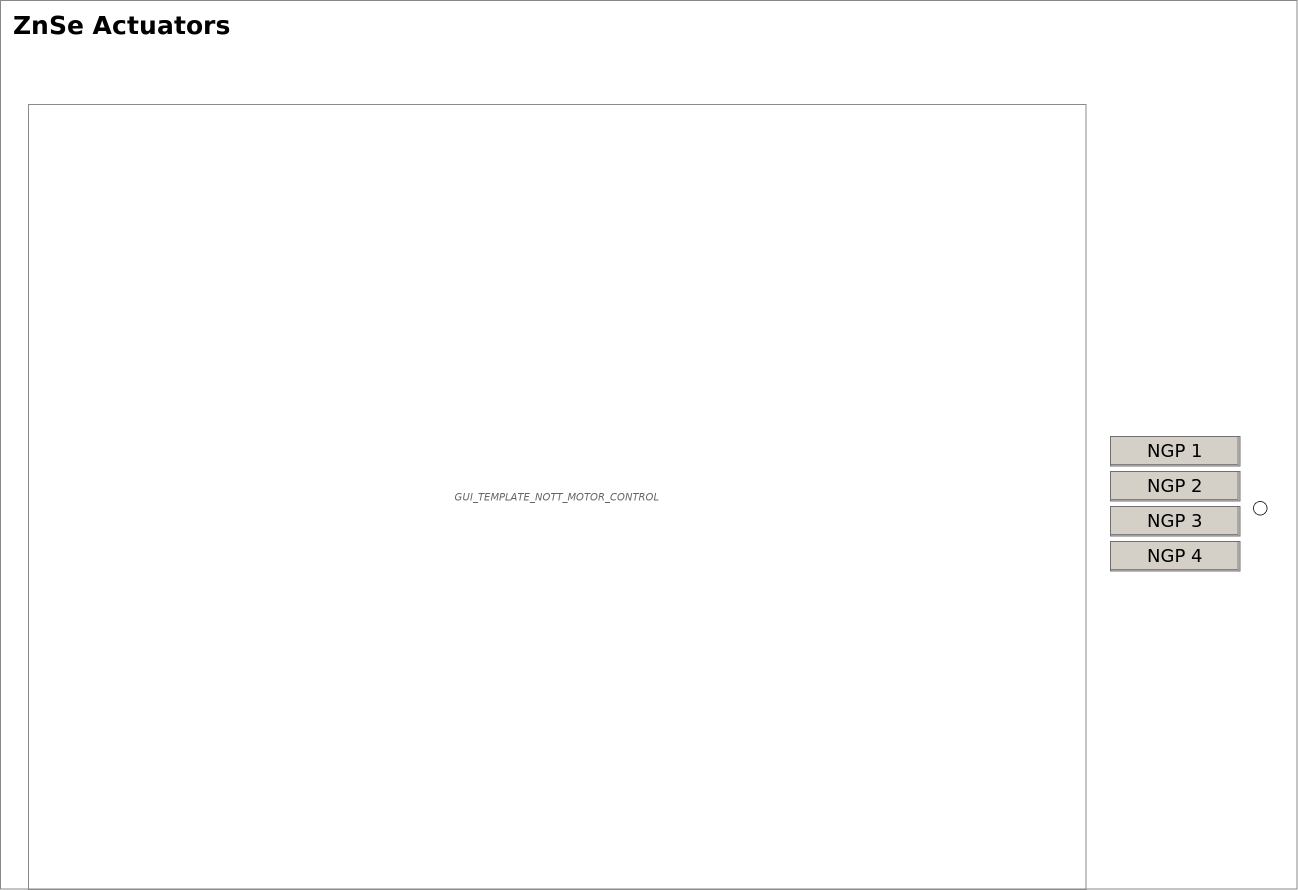
VISUALIZATION VISU_HMI_ZNSE_ACTUATORS  // 1298x890
    Label (10,10 271x30), "ZnSe Actuators"
    Frame (28,104 1058x786)
        shows GUI_TEMPLATE_MOTOR(m_Instance := MAIN.nott_ics.ZnSeActuators.ptrNGPs[MAIN.nott_ics.ZnSeActuators.guiNGPsIndex]^)
    RadioButton (1251,438 47x140), variable: MAIN.nott_ics.ZnSeActuators.guiNGPsIndex-1
        Areas[0]: Text=Radiobutton
        Areas[1]: Text=Radiobutton
    Button (1110,436 130x30), "NGP 1"
        OnMouseClick: execute { MAIN.nott_ics.ZnSeActuators.guiNGPsIndex := 1; }
    Button (1110,471 130x30), "NGP 2"
        OnMouseClick: execute { MAIN.nott_ics.ZnSeActuators.guiNGPsIndex := 2; }
    Button (1110,506 130x30), "NGP 3"
        OnMouseClick: execute { MAIN.nott_ics.ZnSeActuators.guiNGPsIndex := 3; }
    Button (1110,541 130x30), "NGP 4"
        OnMouseClick: execute { MAIN.nott_ics.ZnSeActuators.guiNGPsIndex := 4; }
END_VISUALIZATION

// ---- HMI/VISUs/Templates/CO2_Valve/GUI_TEMPLATE_ACTUATOR_ENG.TcVIS
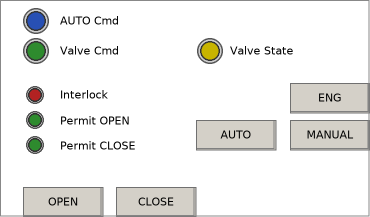
VISUALIZATION GUI_TEMPLATE_ACTUATOR_ENG  // 370x217
VAR_IN_OUT
	m_Cmd:		FB_CRYO_ACTUATOR_CMD;
	m_Valve:	FB_CRYO_VALVE_CTRL;
END_VAR
    Lamp1 (25,85 20x20), variable: m_Cmd.in_bInterlock, style: Lamp-Lamp1-Red
    Lamp1 (25,110 20x20), variable: m_Cmd.bPermitOn, style: Lamp-Lamp1-Green
    Lamp1 (25,135 20x20), variable: m_Cmd.bPermitOff, style: Lamp-Lamp1-Green
    Rectangle (57,80 83x30), "Interlock"
    Rectangle (57,106 83x30), "Permit OPEN"
    Rectangle (57,131 83x30), "Permit CLOSE"
    Button (23,187 80x30), "OPEN", colour toggle: (m_Cmd.bPermitOn AND NOT m_Cmd.bAutoMode) OR m_Cmd.bEngMode, input disabled if: m_Cmd.bDisableBtnOn
        OnMouseClick: execute { m_Cmd.bManualCmd := TRUE; m_Cmd.bManualExecute := TRUE; }
    Lamp1 (21,36 30x30), tooltip "Actual Valve command", variable: m_Cmd.out_bEnable, style: Lamp-Lamp1-Green
    Rectangle (57,36 83x30), "Valve Cmd"
    Button (196,120 80x30), "AUTO", colour toggle: m_Cmd.bAutoMode, input disabled if: m_Cmd.bAutoMode OR m_Cmd.bEngMode
        OnMouseClick: execute { m_Cmd.bAutoMode := TRUE; }
    Button (290,120 80x30), "MANUAL", colour toggle: NOT m_Cmd.bAutoMode, input disabled if: NOT m_Cmd.bAutoMode AND NOT m_Cmd.bEngMode
        OnMouseClick: execute { m_Cmd.bAutoMode := FALSE; }
    Button (116,187 80x30), "CLOSE", colour toggle: (m_Cmd.bPermitOff AND NOT m_Cmd.bAutoMode) OR m_Cmd.bEngMode, input disabled if: m_Cmd.bDisableBtnOff
        OnMouseClick: execute { m_Cmd.bManualCmd := FALSE; m_Cmd.bManualExecute := TRUE; }
    Button (290,83 80x30), "ENG", tooltip "Engineering / Commissioning Mode", colour toggle: m_Cmd.bEngMode, input disabled if: m_Cmd.bAutoMode
        toggle m_Cmd.bEngMode
    Lamp1 (21,6 30x30), tooltip "Command coming from the Control System", variable: m_Cmd.in_bEnable, style: Lamp-Lamp1-Blue
    Rectangle (57,6 83x30), "AUTO Cmd"
    Lamp1 (195,36 30x30), tooltip "Valve state: ON=OPEN, OFF=CLOSED", variable: m_Valve.stat.bActON, style: Lamp-Lamp1-Yellow
    Rectangle (227,36 83x30), "Valve State"
END_VISUALIZATION

// ---- HMI/VISUs/Templates/Motors/GUI_TEMPLATE_MOTOR.TcVIS
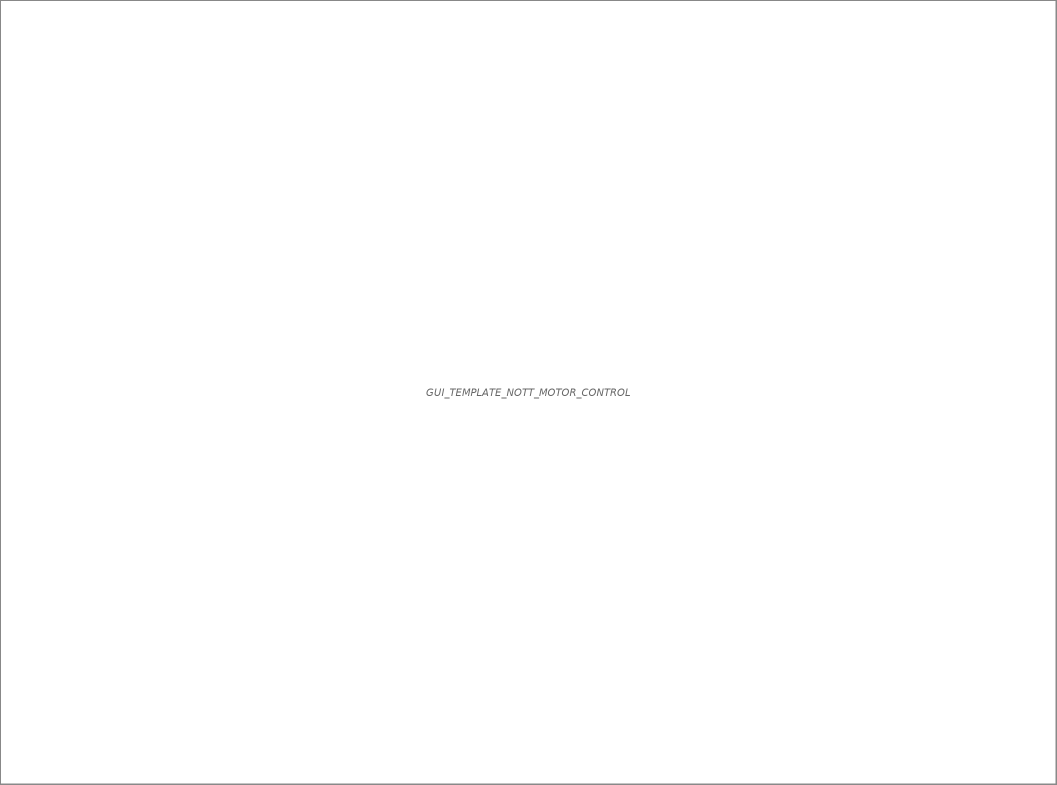
VISUALIZATION GUI_TEMPLATE_MOTOR  // 1057x785
VAR_IN_OUT
	m_Instance:	FB_NOTT_MOTOR;
END_VAR
VAR
	m_lrOffSet : LREAL := 0;
END_VAR
    TabControl (0,0 1057x785)
        shows GUI_TEMPLATE_NOTT_MOTOR_CONTROL(m_Instance := m_Instance)
        shows GUI_TEMPLATE_NOTT_MOTOR_CONFIG(m_Instance := m_Instance)
        [0]: TabTitle=Control
        [1]: TabTitle=Config
END_VISUALIZATION

// ---- HMI/VISUs/Templates/Motors/GUI_TEMPLATE_NOTT_MOTOR_CONFIG.TcVIS
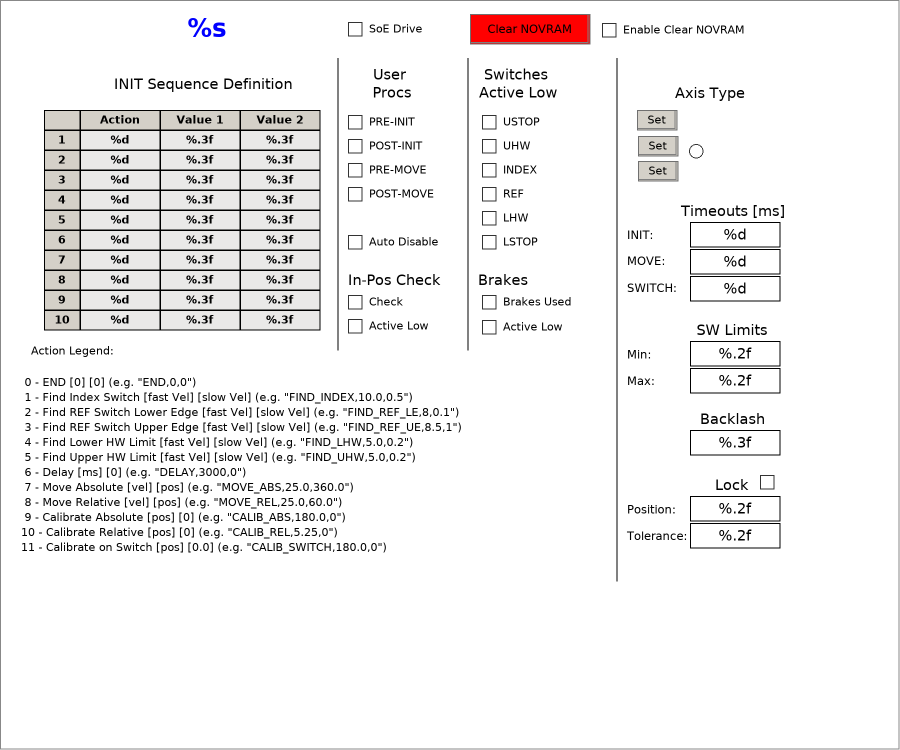
VISUALIZATION GUI_TEMPLATE_NOTT_MOTOR_CONFIG  // 900x750
VAR_IN_OUT
	m_Instance : FB_NOTT_MOTOR;
END_VAR
VAR
	bEnableNovramClear:	BOOL := FALSE;
END_VAR
    Label (28,336 150x30), "Action Legend:"
    Label (18,371 600x23), "0 - END [0] [0] (e.g. "END,0,0")"
    Label (18,386 600x23), "1 - Find Index Switch [fast Vel] [slow Vel] (e.g. "FIND_INDEX,10.0,0.5")"
    Label (18,401 600x23), "2 - Find REF Switch Lower Edge [fast Vel] [slow Vel] (e.g. "FIND_REF_LE,8,0.1")"
    Label (18,416 600x23), "3 - Find REF Switch Upper Edge [fast Vel] [slow Vel] (e.g. "FIND_REF_UE,8.5,1")"
    Label (18,431 600x23), "4 - Find Lower HW Limit [fast Vel] [slow Vel] (e.g. "FIND_LHW,5.0,0.2")"
    Label (18,446 600x23), "5 - Find Upper HW Limit [fast Vel] [slow Vel] (e.g. "FIND_UHW,5.0,0.2")"
    Label (18,476 600x23), "7 - Move Absolute [vel] [pos] (e.g. "MOVE_ABS,25.0,360.0")"
    Label (18,491 600x23), "8 - Move Relative [vel] [pos] (e.g. "MOVE_REL,25.0,60.0")"
    Label (18,506 600x23), "9 - Calibrate Absolute [pos] [0] (e.g. "CALIB_ABS,180.0,0")"
    Label (18,521 600x23), "10 - Calibrate Relative [pos] [0] (e.g. "CALIB_REL,5.25,0")"
    Label (18,461 600x23), "6 - Delay [ms] [0] (e.g. "DELAY,3000,0")"
    Label (18,536 600x23), "11 - Calibrate on Switch [pos] [0.0] (e.g. "CALIB_SWITCH,180.0,0")"
    Label (59,69 289x30), "INIT Sequence Definition"
    Label (462,54 113x59), "Switches Active Low"
    Checkbox (480,110 93x24), "USTOP", variable: m_Instance.cfg.bArrActiveLow[5].bValue, invisible if: false, input disabled if: false
    Checkbox (480,134 93x24), "UHW", variable: m_Instance.cfg.bArrActiveLow[4].bValue, invisible if: false, input disabled if: false
    Checkbox (480,158 93x24), "INDEX", variable: m_Instance.cfg.bArrActiveLow[3].bValue, invisible if: false, input disabled if: false
    Checkbox (480,182 93x24), "REF", variable: m_Instance.cfg.bArrActiveLow[2].bValue, invisible if: false, input disabled if: false
    Checkbox (480,206 93x24), "LHW", variable: m_Instance.cfg.bArrActiveLow[1].bValue, invisible if: false, input disabled if: false
    Checkbox (480,230 93x24), "LSTOP", variable: m_Instance.cfg.bArrActiveLow[0].bValue, invisible if: false, input disabled if: false
    Rectangle (87,7 240x42), "%s", text variable: m_Instance.sName
    Label (678,196 132x30), "Timeouts [ms]"
    Label (665,78 90x30), "Axis Type"
    Label (687,315 90x30), "SW Limits"
    Label (475,265 103x30), "Brakes"
    Label (685,404 95x30), "Backlash"
    RadioButton (687,112 114x78), variable: m_Instance.cfg.nAxisType-1, input disabled if: FALSE
        Areas[0]: Text=Linear
        Areas[1]: Text=Circular
        Areas[2]: Text=Circular-Opt
        p3166011961: Cicular-Optimised
    Checkbox (480,290 110x24), "Brakes Used", variable: m_Instance.cfg.bUseBrake, invisible if: false, input disabled if: false
    Checkbox (480,315 105x24), "Active Low", tooltip "Brake Feedback Signal is Active Low", variable: m_Instance.cfg.bActiveLowBrake, invisible if: false, input disabled if: false
    Rectangle (690,430 90x25), "%.3f", tooltip "Positive, negative or zero (no backlash)", text variable: m_Instance.cfg.lrBacklash
        OnMouseDown: write the text variable via Default
    Button (637,110 40x20), "Set"
        OnMouseClick: execute { m_Instance.cfg.nAxisType := 1; }
    Button (638,136 40x20), "Set"
        OnMouseClick: execute { m_Instance.cfg.nAxisType := 2; }
    Button (638,161 40x20), "Set"
        OnMouseClick: execute { m_Instance.cfg.nAxisType := 3; }
    Rectangle (690,341 90x25), "%.2f", tooltip "Setting both limits to 0 means that limits are not used.", text variable: m_Instance.cfg.lrMinPosition
        OnMouseDown: write the text variable via Default
    Rectangle (690,368 90x25), "%.2f", tooltip "Setting both limits to 0 means that limits are not used.", text variable: m_Instance.cfg.lrMaxPosition
        OnMouseDown: write the text variable via Default
    Label (624,340 37x29), "Min:"
    Label (624,366 37x30), "Max:"
    Label (624,220 49x30), "INIT:"
    Label (624,246 49x30), "MOVE:"
    Rectangle (690,222 90x25), "%d", tooltip "INIT sequence timeout in [ms].", text variable: m_Instance.cfg.nTimeoutInit
        OnMouseDown: write the text variable via Default
    Rectangle (690,249 90x25), "%d", tooltip "INIT sequence timeout in [ms].", text variable: m_Instance.cfg.nTimeoutMove
        OnMouseDown: write the text variable via Default
    Line (468,350) (468,58)
    Line (617,581) (617,58)
    Rectangle (690,276 90x25), "%d", tooltip "Switch exit timeout in [ms].", text variable: m_Instance.cfg.nTimeoutSwitch
        OnMouseDown: write the text variable via Default
    Label (624,273 60x30), "SWITCH:"
    Rectangle (80,110 80x20), "Action"
    Rectangle (160,110 80x20), "Value 1"
    Rectangle (240,110 80x20), "Value 2"
    Rectangle (44,130 36x20), "1"
    Rectangle (44,110 36x20)
    Rectangle (80,130 80x20), "%d", text variable: m_Instance.cfg.strArrInitSeq[1].nAction
        OnMouseDown: write the text variable via Default
    Rectangle (160,130 80x20), "%.3f", text variable: m_Instance.cfg.strArrInitSeq[1].lrValue1
        OnMouseDown: write the text variable via Default
    Rectangle (240,130 80x20), "%.3f", text variable: m_Instance.cfg.strArrInitSeq[1].lrValue2
        OnMouseDown: write the text variable via Default
    Rectangle (44,150 36x20), "2"
    Rectangle (80,150 80x20), "%d", text variable: m_Instance.cfg.strArrInitSeq[2].nAction
        OnMouseDown: write the text variable via Default
    Rectangle (160,150 80x20), "%.3f", text variable: m_Instance.cfg.strArrInitSeq[2].lrValue1
        OnMouseDown: write the text variable via Default
    Rectangle (240,150 80x20), "%.3f", text variable: m_Instance.cfg.strArrInitSeq[2].lrValue2
        OnMouseDown: write the text variable via Default
    Rectangle (44,170 36x20), "3"
    Rectangle (80,170 80x20), "%d", text variable: m_Instance.cfg.strArrInitSeq[3].nAction
        OnMouseDown: write the text variable via Default
    Rectangle (160,170 80x20), "%.3f", text variable: m_Instance.cfg.strArrInitSeq[3].lrValue1
        OnMouseDown: write the text variable via Default
    Rectangle (240,170 80x20), "%.3f", text variable: m_Instance.cfg.strArrInitSeq[3].lrValue2
        OnMouseDown: write the text variable via Default
    Rectangle (44,190 36x20), "4"
    Rectangle (80,190 80x20), "%d", text variable: m_Instance.cfg.strArrInitSeq[4].nAction
        OnMouseDown: write the text variable via Default
    Rectangle (160,190 80x20), "%.3f", text variable: m_Instance.cfg.strArrInitSeq[4].lrValue1
        OnMouseDown: write the text variable via Default
    Rectangle (240,190 80x20), "%.3f", text variable: m_Instance.cfg.strArrInitSeq[4].lrValue2
        OnMouseDown: write the text variable via Default
    Rectangle (44,210 36x20), "5"
    Rectangle (80,210 80x20), "%d", text variable: m_Instance.cfg.strArrInitSeq[5].nAction
        OnMouseDown: write the text variable via Default
    Rectangle (160,210 80x20), "%.3f", text variable: m_Instance.cfg.strArrInitSeq[5].lrValue1
        OnMouseDown: write the text variable via Default
    Rectangle (240,210 80x20), "%.3f", text variable: m_Instance.cfg.strArrInitSeq[5].lrValue2
        OnMouseDown: write the text variable via Default
    Rectangle (44,230 36x20), "6"
    Rectangle (80,230 80x20), "%d", text variable: m_Instance.cfg.strArrInitSeq[6].nAction
        OnMouseDown: write the text variable via Default
    Rectangle (160,230 80x20), "%.3f", text variable: m_Instance.cfg.strArrInitSeq[6].lrValue1
        OnMouseDown: write the text variable via Default
    Rectangle (240,230 80x20), "%.3f", text variable: m_Instance.cfg.strArrInitSeq[6].lrValue2
        OnMouseDown: write the text variable via Default
    Rectangle (44,250 36x20), "7"
    Rectangle (80,250 80x20), "%d", text variable: m_Instance.cfg.strArrInitSeq[7].nAction
        OnMouseDown: write the text variable via Default
    Rectangle (160,250 80x20), "%.3f", text variable: m_Instance.cfg.strArrInitSeq[7].lrValue1
        OnMouseDown: write the text variable via Default
    Rectangle (240,250 80x20), "%.3f", text variable: m_Instance.cfg.strArrInitSeq[7].lrValue2
        OnMouseDown: write the text variable via Default
    Rectangle (44,270 36x20), "8"
    Rectangle (80,270 80x20), "%d", text variable: m_Instance.cfg.strArrInitSeq[8].nAction
        OnMouseDown: write the text variable via Default
    Rectangle (160,270 80x20), "%.3f", text variable: m_Instance.cfg.strArrInitSeq[8].lrValue1
        OnMouseDown: write the text variable via Default
    Rectangle (240,270 80x20), "%.3f", text variable: m_Instance.cfg.strArrInitSeq[8].lrValue2
        OnMouseDown: write the text variable via Default
    Rectangle (44,290 36x20), "9"
    Rectangle (80,290 80x20), "%d", text variable: m_Instance.cfg.strArrInitSeq[9].nAction
        OnMouseDown: write the text variable via Default
    Rectangle (160,290 80x20), "%.3f", text variable: m_Instance.cfg.strArrInitSeq[9].lrValue1
        OnMouseDown: write the text variable via Default
    Rectangle (240,290 80x20), "%.3f", text variable: m_Instance.cfg.strArrInitSeq[9].lrValue2
        OnMouseDown: write the text variable via Default
    Rectangle (44,310 36x20), "10"
    Rectangle (80,310 80x20), "%d", text variable: m_Instance.cfg.strArrInitSeq[10].nAction
        OnMouseDown: write the text variable via Default
    Rectangle (160,310 80x20), "%.3f", text variable: m_Instance.cfg.strArrInitSeq[10].lrValue1
        OnMouseDown: write the text variable via Default
    Rectangle (240,310 80x20), "%.3f", text variable: m_Instance.cfg.strArrInitSeq[10].lrValue2
        OnMouseDown: write the text variable via Default
    Line (338,350) (338,58)
    Label (345,54 94x59), "User Procs"
    Checkbox (346,110 106x24), "PRE-INIT", variable: m_Instance.cfg.bExecUserPreInit, invisible if: false, input disabled if: false
    Checkbox (346,134 106x24), "POST-INIT", variable: m_Instance.cfg.bExecUserPostInit, invisible if: false, input disabled if: false
    Checkbox (346,158 106x24), "PRE-MOVE", variable: m_Instance.cfg.bExecUserPreMove, invisible if: false, input disabled if: false
    Checkbox (346,182 106x24), "POST-MOVE", variable: m_Instance.cfg.bExecUserPostMove, invisible if: false, input disabled if: false
    Label (687,470 90x30), "Lock"
    Rectangle (690,496 90x25), "%.2f", tooltip "If the motor is locked, during INIT the motor will not move and its position will be set to this value.", text variable: m_Instance.cfg.lrLockPos
        OnMouseDown: write the text variable via Default
    Rectangle (690,523 90x25), "%.2f", tooltip "The motor will not move, if the target position is closer to the locked position than this value.", text variable: m_Instance.cfg.lrLockTol
        OnMouseDown: write the text variable via Default
    Label (624,495 56x29), "Position:"
    Label (624,521 63x30), "Tolerance:"
    Checkbox (758,470 30x24), tooltip "Flag if motor is locked", variable: m_Instance.cfg.bLock, invisible if: false, input disabled if: false
    Checkbox (346,290 106x24), "Check", tooltip "If active, check if the in-pos signal is active after the move completes. If it is not, it's a failure.", variable: m_Instance.cfg.bCheckInPos, invisible if: false, input disabled if: false
    Checkbox (346,314 107x24), "Active Low", tooltip "If checked, In-Position feedback signal is active low", variable: m_Instance.cfg.bActiveLowInPos, invisible if: false, input disabled if: false
    Checkbox (346,230 127x24), "Auto Disable", tooltip "Auto Disable Motor After Move", variable: m_Instance.cfg.bDisableAfterMove, invisible if: false, input disabled if: false
    Label (345,265 103x30), "In-Pos Check"
    Button (470,14 120x30), "Clear NOVRAM", tooltip "Clear NOVRAM. Use it with care! This is needed ONLY if NOVRAM was previously used for data structures different than T_MOTOR_CFG (or for previous versions of T_MOTOR_CFG). Bring the motor to NOT_READY first and then clear NOVRAM.", input disabled if: bEnableNovramClear=false OR m_Instance.nNOVRAM_DevId=0
        OnMouseUp: execute {
            m_Instance.ctrl.bLocalCmd := TRUE;
            m_Instance.ctrl.nCommand:=E_MOTOR_COMMAND.CLEAR_NOVRAM;
            m_Instance.ctrl.bExecute:=(TRUE);
        }
    Checkbox (600,18 160x24), "Enable Clear NOVRAM", variable: bEnableNovramClear, invisible if: false, input disabled if: false
    Checkbox (346,17 90x24), "SoE Drive", tooltip "Check the box if this is an SoE drive (Sercos over EtherCAT) , e.g. AX5000", variable: m_Instance.cfg.bSoE_Drive, invisible if: false, input disabled if: false
END_VISUALIZATION

